Universal Robots PolyScope program: inkscape-test-1.urp

Program inkscape-test-1 (installation=default directory=/programs createdIn=5.11.9.1010452 lastSavedIn=5.11.9.1010452 robotSerialNumber=20225200364)
Calibrated DH parameters: a=[0.00002, -0.569483, -0.54992, -0.00001, -0.000036, 0]; d=[0.180894, -146.691669, 192.918669, -46.053088, 0.119778, 0.115602]; alpha=[1.571425, -0.001534, 0.003359, 1.568739, -1.571477, 0]; deltaTheta=[0, 0.376258, -0.101074, -0.275185, -0.000002, 0]
Robot Program (runOnlyOnce=true)
  Script file /programs/usbdisk/robot_new_inkscape_test_9.script
    | def Machining3():
    |   # Default parameters:
    |   global speed_ms = 0.3
    |   global speed_rads = 0.75
    |   global accel_mss = 3
    |   global accel_radss = 1.2
    |   global blend_radius_m = 0.001
    | 
    |   # Add subprograms here
    |   # Start of main program
    |   # Program generated by RoboDK v5.6.5 for UR10e on 16/10/2023 17:33:41
    |   # Using nominal kinematics.
    |   blend_radius_m = 0.001
    |   speed_ms = 1.000
    |   # set_reference(p[0.335000, -0.154000, -0.015800, 0.000000, 0.000000, 0.000000])
    |   set_tcp(p[0.000000, 0.000000, 0.252000, 0.000000, 0.000000, 0.000000])
    |   # Show Tool
    |   movej([0.061043, -1.073805, -2.582860, -1.055724, 1.570796, 1.631840],accel_radss,speed_rads,0,blend_radius_m)
    |   movel([0.061043, -1.164815, -2.648932, -0.898642, 1.570796, 1.631840],accel_mss,speed_ms,0,blend_radius_m)
    |   speed_ms = 1.000
    |   speed_ms = 0.005
    |   movel([0.061043, -1.124589, -2.623317, -0.964483, 1.570796, 1.631840],accel_mss,speed_ms,0,blend_radius_m)
    |   speed_ms = 1.000
    |   movel([0.061043, -1.164815, -2.648932, -0.898642, 1.570796, 1.631840],accel_mss,speed_ms,0,blend_radius_m)
    |   speed_ms = 0.040
    |   speed_ms = 1.000
    |   movel([0.120277, -1.219092, -2.622470, -0.870827, 1.570796, 1.691073],accel_mss,speed_ms,0,blend_radius_m)
    |   speed_ms = 0.005
    |   movel([0.120277, -1.264094, -2.645638, -0.802657, 1.570796, 1.691073],accel_mss,speed_ms,0,blend_radius_m)
    |   speed_ms = 0.030
    |   movel([0.129753, -1.261000, -2.647334, -0.804055, 1.570796, 1.700549],accel_mss,speed_ms,0,blend_radius_m)
    |   movel([0.141933, -1.256916, -2.649554, -0.805919, 1.570796, 1.712729],accel_mss,speed_ms,0,blend_radius_m)
    |   movel([0.142238, -1.256582, -2.649735, -0.806073, 1.570796, 1.713034],accel_mss,speed_ms,0,blend_radius_m)
    |   movel([0.142012, -1.256413, -2.649826, -0.806150, 1.570796, 1.712808],accel_mss,speed_ms,0,blend_radius_m)
    |   movel([0.136669, -1.257955, -2.648991, -0.805443, 1.570796, 1.707466],accel_mss,speed_ms,0,blend_radius_m)
    |   movel([0.120416, -1.263053, -2.646210, -0.803126, 1.570796, 1.691212],accel_mss,speed_ms,0,blend_radius_m)
    |   movel([0.110953, -1.266208, -2.644473, -0.801708, 1.570796, 1.681749],accel_mss,speed_ms,0,blend_radius_m)
    |   movel([0.098869, -1.270513, -2.642083, -0.799793, 1.570796, 1.669665],accel_mss,speed_ms,0,blend_radius_m)
    |   movel([0.098580, -1.270845, -2.641898, -0.799646, 1.570796, 1.669376],accel_mss,speed_ms,0,blend_radius_m)
    |   movel([0.098815, -1.270997, -2.641813, -0.799579, 1.570796, 1.669612],accel_mss,speed_ms,0,blend_radius_m)
    |   movel([0.104107, -1.269335, -2.642739, -0.800314, 1.570796, 1.674903],accel_mss,speed_ms,0,blend_radius_m)
    |   movel([0.120277, -1.264094, -2.645638, -0.802657, 1.570796, 1.691073],accel_mss,speed_ms,0,blend_radius_m)
    |   movel([0.123150, -1.263148, -2.646158, -0.803083, 1.570796, 1.693947],accel_mss,speed_ms,0,blend_radius_m)
    |   speed_ms = 0.005
    |   movel([0.123150, -1.253718, -2.641632, -0.817039, 1.570796, 1.693947],accel_mss,speed_ms,0,blend_radius_m)
    |   speed_ms = 0.040
    |   movel([0.120555, -1.252576, -2.642250, -0.817563, 1.570796, 1.691351],accel_mss,speed_ms,0,blend_radius_m)
    |   speed_ms = 0.005
    |   movel([0.120555, -1.262011, -2.646781, -0.803597, 1.570796, 1.691351],accel_mss,speed_ms,0,blend_radius_m)
    |   speed_ms = 0.030
    |   movel([0.142487, -1.254991, -2.650593, -0.806805, 1.570796, 1.713283],accel_mss,speed_ms,0,blend_radius_m)
    |   movel([0.142694, -1.253662, -2.651308, -0.807419, 1.570796, 1.713491],accel_mss,speed_ms,0,blend_radius_m)
    |   movel([0.142903, -1.252330, -2.652023, -0.808036, 1.570796, 1.713699],accel_mss,speed_ms,0,blend_radius_m)
    |   movel([0.120905, -1.259399, -2.648206, -0.804783, 1.570796, 1.691701],accel_mss,speed_ms,0,blend_radius_m)
    |   movel([0.099033, -1.266750, -2.644174, -0.801466, 1.570796, 1.669830],accel_mss,speed_ms,0,blend_radius_m)
    |   movel([0.098891, -1.268032, -2.643463, -0.800894, 1.570796, 1.669687],accel_mss,speed_ms,0,blend_radius_m)
    |   movel([0.098749, -1.269312, -2.642752, -0.800325, 1.570796, 1.669546],accel_mss,speed_ms,0,blend_radius_m)
    |   movel([0.120555, -1.262011, -2.646781, -0.803597, 1.570796, 1.691351],accel_mss,speed_ms,0,blend_radius_m)
    |   movel([0.123434, -1.261071, -2.647295, -0.804023, 1.570796, 1.694230],accel_mss,speed_ms,0,blend_radius_m)
    |   speed_ms = 0.005
    |   movel([0.123434, -1.251631, -2.642760, -0.817998, 1.570796, 1.694230],accel_mss,speed_ms,0,blend_radius_m)
    |   speed_ms = 0.040
    |   movel([0.121045, -1.248898, -2.644228, -0.819263, 1.570796, 1.691842],accel_mss,speed_ms,0,blend_radius_m)
    |   speed_ms = 0.005
    |   movel([0.121045, -1.258351, -2.648776, -0.805262, 1.570796, 1.691842],accel_mss,speed_ms,0,blend_radius_m)
    |   speed_ms = 0.030
    |   movel([0.106723, -1.263119, -2.646174, -0.803096, 1.570796, 1.677520],accel_mss,speed_ms,0,blend_radius_m)
    |   movel([0.102037, -1.264600, -2.645360, -0.802429, 1.570796, 1.672833],accel_mss,speed_ms,0,blend_radius_m)
    |   movel([0.099769, -1.265127, -2.645070, -0.802192, 1.570796, 1.670566],accel_mss,speed_ms,0,blend_radius_m)
    |   movel([0.099380, -1.265045, -2.645115, -0.802229, 1.570796, 1.670177],accel_mss,speed_ms,0,blend_radius_m)
    |   movel([0.099262, -1.264692, -2.645309, -0.802388, 1.570796, 1.670058],accel_mss,speed_ms,0,blend_radius_m)
    |   movel([0.099472, -1.264226, -2.645566, -0.802597, 1.570796, 1.670268],accel_mss,speed_ms,0,blend_radius_m)
    |   movel([0.099911, -1.263859, -2.645767, -0.802763, 1.570796, 1.670707],accel_mss,speed_ms,0,blend_radius_m)
    |   movel([0.102241, -1.262808, -2.646345, -0.803237, 1.570796, 1.673038],accel_mss,speed_ms,0,blend_radius_m)
    |   movel([0.106966, -1.261080, -2.647290, -0.804019, 1.570796, 1.677763],accel_mss,speed_ms,0,blend_radius_m)
    |   movel([0.121327, -1.256251, -2.649914, -0.806225, 1.570796, 1.692123],accel_mss,speed_ms,0,blend_radius_m)
    |   movel([0.135738, -1.251578, -2.652425, -0.808386, 1.570796, 1.706534],accel_mss,speed_ms,0,blend_radius_m)
    |   movel([0.140472, -1.250185, -2.653169, -0.809035, 1.570796, 1.711269],accel_mss,speed_ms,0,blend_radius_m)
    |   movel([0.142756, -1.249719, -2.653417, -0.809253, 1.570796, 1.713552],accel_mss,speed_ms,0,blend_radius_m)
    |   movel([0.143139, -1.249820, -2.653363, -0.809206, 1.570796, 1.713935],accel_mss,speed_ms,0,blend_radius_m)
    |   movel([0.143238, -1.250193, -2.653165, -0.809031, 1.570796, 1.714034],accel_mss,speed_ms,0,blend_radius_m)
    |   movel([0.143005, -1.250671, -2.652910, -0.808808, 1.570796, 1.713802],accel_mss,speed_ms,0,blend_radius_m)
    |   movel([0.142550, -1.251035, -2.652715, -0.808639, 1.570796, 1.713347],accel_mss,speed_ms,0,blend_radius_m)
    |   movel([0.140187, -1.252037, -2.652180, -0.808172, 1.570796, 1.710984],accel_mss,speed_ms,0,blend_radius_m)
    |   movel([0.135426, -1.253668, -2.651305, -0.807416, 1.570796, 1.706223],accel_mss,speed_ms,0,blend_radius_m)
    |   movel([0.121045, -1.258351, -2.648776, -0.805262, 1.570796, 1.691842],accel_mss,speed_ms,0,blend_radius_m)
    |   movel([0.118157, -1.259303, -2.648259, -0.804827, 1.570796, 1.688953],accel_mss,speed_ms,0,blend_radius_m)
    |   speed_ms = 0.005
    |   movel([0.118157, -1.249854, -2.643716, -0.818819, 1.570796, 1.688953],accel_mss,speed_ms,0,blend_radius_m)
    |   speed_ms = 0.040
    |   movel([0.121469, -1.245729, -2.645920, -0.820740, 1.570796, 1.692265],accel_mss,speed_ms,0,blend_radius_m)
    |   speed_ms = 0.005
    |   movel([0.121469, -1.255197, -2.650482, -0.806710, 1.570796, 1.692265],accel_mss,speed_ms,0,blend_radius_m)
    |   speed_ms = 0.030
    |   movel([0.105133, -1.260563, -2.647572, -0.804254, 1.570796, 1.675929],accel_mss,speed_ms,0,blend_radius_m)
    |   movel([0.099787, -1.262265, -2.646642, -0.803482, 1.570796, 1.670583],accel_mss,speed_ms,0,blend_radius_m)
    |   movel([0.099549, -1.262111, -2.646726, -0.803552, 1.570796, 1.670346],accel_mss,speed_ms,0,blend_radius_m)
    |   movel([0.099842, -1.261774, -2.646911, -0.803704, 1.570796, 1.670638],accel_mss,speed_ms,0,blend_radius_m)
    |   movel([0.112050, -1.257371, -2.649308, -0.805711, 1.570796, 1.682846],accel_mss,speed_ms,0,blend_radius_m)
    |   movel([0.121610, -1.254143, -2.651050, -0.807196, 1.570796, 1.692407],accel_mss,speed_ms,0,blend_radius_m)
    |   movel([0.138032, -1.248922, -2.653841, -0.809626, 1.570796, 1.708829],accel_mss,speed_ms,0,blend_radius_m)
    |   movel([0.143430, -1.247342, -2.654680, -0.810368, 1.570796, 1.714226],accel_mss,speed_ms,0,blend_radius_m)
    |   movel([0.143659, -1.247512, -2.654589, -0.810288, 1.570796, 1.714455],accel_mss,speed_ms,0,blend_radius_m)
    |   movel([0.143350, -1.247852, -2.654409, -0.810128, 1.570796, 1.714146],accel_mss,speed_ms,0,blend_radius_m)
    |   movel([0.131042, -1.252031, -2.652183, -0.808175, 1.570796, 1.701839],accel_mss,speed_ms,0,blend_radius_m)
    |   movel([0.121469, -1.255197, -2.650482, -0.806710, 1.570796, 1.692265],accel_mss,speed_ms,0,blend_radius_m)
    |   movel([0.118572, -1.256136, -2.649976, -0.806278, 1.570796, 1.689369],accel_mss,speed_ms,0,blend_radius_m)
    |   speed_ms = 0.005
    |   movel([0.118572, -1.246672, -2.645418, -0.820299, 1.570796, 1.689369],accel_mss,speed_ms,0,blend_radius_m)
    |   speed_ms = 0.040
    |   movel([0.121895, -1.242544, -2.647608, -0.822237, 1.570796, 1.692691],accel_mss,speed_ms,0,blend_radius_m)
    |   speed_ms = 0.005
    |   movel([0.121895, -1.252028, -2.652185, -0.808177, 1.570796, 1.692691],accel_mss,speed_ms,0,blend_radius_m)
    |   speed_ms = 0.030
    |   movel([0.099260, -1.259721, -2.648031, -0.804637, 1.570796, 1.670056],accel_mss,speed_ms,0,blend_radius_m)
    |   movel([0.101199, -1.242362, -2.657302, -0.812725, 1.570796, 1.671995],accel_mss,speed_ms,0,blend_radius_m)
    |   movel([0.103217, -1.224523, -2.666459, -0.821407, 1.570796, 1.674013],accel_mss,speed_ms,0,blend_radius_m)
    |   movel([0.126797, -1.216082, -2.670663, -0.825644, 1.570796, 1.697593],accel_mss,speed_ms,0,blend_radius_m)
    |   movel([0.150532, -1.207955, -2.674635, -0.829799, 1.570796, 1.721329],accel_mss,speed_ms,0,blend_radius_m)
    |   movel([0.147540, -1.226560, -2.665432, -0.820397, 1.570796, 1.718336],accel_mss,speed_ms,0,blend_radius_m)
    |   movel([0.144667, -1.244634, -2.656110, -0.811646, 1.570796, 1.715464],accel_mss,speed_ms,0,blend_radius_m)
    |   movel([0.121895, -1.252028, -2.652185, -0.808177, 1.570796, 1.692691],accel_mss,speed_ms,0,blend_radius_m)
    |   movel([0.118985, -1.252998, -2.651665, -0.807726, 1.570796, 1.689781],accel_mss,speed_ms,0,blend_radius_m)
    |   speed_ms = 0.005
    |   movel([0.118985, -1.243519, -2.647093, -0.821777, 1.570796, 1.689781],accel_mss,speed_ms,0,blend_radius_m)
    |   speed_ms = 0.040
    |   movel([0.126726, -1.204862, -2.666692, -0.840834, 1.570796, 1.697522],accel_mss,speed_ms,0,blend_radius_m)
    |   speed_ms = 0.005
    |   movel([0.126726, -1.214506, -2.671439, -0.826444, 1.570796, 1.697522],accel_mss,speed_ms,0,blend_radius_m)
    |   speed_ms = 0.030
    |   movel([0.104008, -1.222655, -2.667396, -0.822338, 1.570796, 1.674804],accel_mss,speed_ms,0,blend_radius_m)
    |   movel([0.105123, -1.212962, -2.672197, -0.827230, 1.570796, 1.675919],accel_mss,speed_ms,0,blend_radius_m)
    |   movel([0.106263, -1.203120, -2.676963, -0.832306, 1.570796, 1.677059],accel_mss,speed_ms,0,blend_radius_m)
    |   movel([0.129497, -1.194544, -2.681029, -0.836816, 1.570796, 1.700293],accel_mss,speed_ms,0,blend_radius_m)
    |   movel([0.152886, -1.186265, -2.684878, -0.841246, 1.570796, 1.723683],accel_mss,speed_ms,0,blend_radius_m)
    |   movel([0.151219, -1.196537, -2.680091, -0.835761, 1.570796, 1.722015],accel_mss,speed_ms,0,blend_radius_m)
    |   movel([0.149588, -1.206647, -2.675268, -0.830475, 1.570796, 1.720384],accel_mss,speed_ms,0,blend_radius_m)
    |   movel([0.126726, -1.214506, -2.671439, -0.826444, 1.570796, 1.697522],accel_mss,speed_ms,0,blend_radius_m)
    |   movel([0.123688, -1.215576, -2.670913, -0.825900, 1.570796, 1.694484],accel_mss,speed_ms,0,blend_radius_m)
    |   speed_ms = 0.005
    |   movel([0.123688, -1.205937, -2.666170, -0.840282, 1.570796, 1.694484],accel_mss,speed_ms,0,blend_radius_m)
    |   speed_ms = 0.040
    |   movel([0.157276, -1.164256, -2.685501, -0.862631, 1.570796, 1.728073],accel_mss,speed_ms,0,blend_radius_m)
    |   speed_ms = 0.005
    |   movel([0.157276, -1.174031, -2.690432, -0.847927, 1.570796, 1.728073],accel_mss,speed_ms,0,blend_radius_m)
    |   speed_ms = 0.030
    |   movel([0.255784, -1.142912, -2.703858, -0.865619, 1.570796, 1.826580],accel_mss,speed_ms,0,blend_radius_m)
    |   movel([0.213690, -1.314067, -2.616588, -0.781734, 1.570796, 1.784487],accel_mss,speed_ms,0,blend_radius_m)
    |   movel([0.183803, -1.448210, -2.521691, -0.742489, 1.570796, 1.754599],accel_mss,speed_ms,0,blend_radius_m)
    |   movel([0.113774, -1.462570, -2.509956, -0.739863, 1.570796, 1.684571],accel_mss,speed_ms,0,blend_radius_m)
    |   movel([0.044558, -1.480296, -2.495031, -0.737062, 1.570796, 1.615354],accel_mss,speed_ms,0,blend_radius_m)
    |   movel([0.051500, -1.358795, -2.587796, -0.765798, 1.570796, 1.622297],accel_mss,speed_ms,0,blend_radius_m)
    |   movel([0.061043, -1.210716, -2.673294, -0.828379, 1.570796, 1.631840],accel_mss,speed_ms,0,blend_radius_m)
    |   movel([0.157276, -1.174031, -2.690432, -0.847927, 1.570796, 1.728073],accel_mss,speed_ms,0,blend_radius_m)
    |   movel([0.160447, -1.172924, -2.690926, -0.848539, 1.570796, 1.731244],accel_mss,speed_ms,0,blend_radius_m)
    |   speed_ms = 0.005
    |   movel([0.160447, -1.163146, -2.685991, -0.863252, 1.570796, 1.731244],accel_mss,speed_ms,0,blend_radius_m)
    |   speed_ms = 0.040
    |   movel([0.178723, -1.187438, -2.674979, -0.849972, 1.570796, 1.749519],accel_mss,speed_ms,0,blend_radius_m)
    |   speed_ms = 0.005
    |   movel([0.178723, -1.197143, -2.679805, -0.835441, 1.570796, 1.749519],accel_mss,speed_ms,0,blend_radius_m)
    |   speed_ms = 0.030
    |   movel([0.155706, -1.204603, -2.676252, -0.831534, 1.570796, 1.726503],accel_mss,speed_ms,0,blend_radius_m)
    |   movel([0.157407, -1.194439, -2.681078, -0.836872, 1.570796, 1.728204],accel_mss,speed_ms,0,blend_radius_m)
    |   movel([0.159147, -1.184110, -2.685868, -0.842411, 1.570796, 1.729943],accel_mss,speed_ms,0,blend_radius_m)
    |   movel([0.182702, -1.176243, -2.689439, -0.846707, 1.570796, 1.753498],accel_mss,speed_ms,0,blend_radius_m)
    |   movel([0.206362, -1.168729, -2.692789, -0.850871, 1.570796, 1.777158],accel_mss,speed_ms,0,blend_radius_m)
    |   movel([0.204073, -1.179467, -2.687983, -0.844938, 1.570796, 1.774869],accel_mss,speed_ms,0,blend_radius_m)
    |   movel([0.201836, -1.190024, -2.683139, -0.839225, 1.570796, 1.772633],accel_mss,speed_ms,0,blend_radius_m)
    |   movel([0.178723, -1.197143, -2.679805, -0.835441, 1.570796, 1.749519],accel_mss,speed_ms,0,blend_radius_m)
    |   movel([0.175648, -1.198119, -2.679344, -0.834926, 1.570796, 1.746444],accel_mss,speed_ms,0,blend_radius_m)
    |   speed_ms = 0.005
    |   movel([0.175648, -1.188417, -2.674523, -0.849450, 1.570796, 1.746444],accel_mss,speed_ms,0,blend_radius_m)
    |   speed_ms = 0.040
    |   movel([0.170964, -1.226858, -2.655750, -0.829781, 1.570796, 1.741760],accel_mss,speed_ms,0,blend_radius_m)
    |   speed_ms = 0.005
    |   movel([0.170964, -1.236412, -2.660397, -0.815579, 1.570796, 1.741760],accel_mss,speed_ms,0,blend_radius_m)
    |   speed_ms = 0.030
    |   movel([0.193490, -1.230002, -2.663685, -0.818701, 1.570796, 1.764287],accel_mss,speed_ms,0,blend_radius_m)
    |   movel([0.197334, -1.211473, -2.672925, -0.827991, 1.570796, 1.768131],accel_mss,speed_ms,0,blend_radius_m)
    |   movel([0.199301, -1.201920, -2.677537, -0.832932, 1.570796, 1.770097],accel_mss,speed_ms,0,blend_radius_m)
    |   movel([0.200933, -1.192747, -2.681871, -0.837771, 1.570796, 1.771729],accel_mss,speed_ms,0,blend_radius_m)
    |   movel([0.200878, -1.192448, -2.682010, -0.837931, 1.570796, 1.771674],accel_mss,speed_ms,0,blend_radius_m)
    |   movel([0.200628, -1.192319, -2.682071, -0.837999, 1.570796, 1.771424],accel_mss,speed_ms,0,blend_radius_m)
    |   movel([0.200026, -1.192393, -2.682036, -0.837960, 1.570796, 1.770823],accel_mss,speed_ms,0,blend_radius_m)
    |   movel([0.177133, -1.199429, -2.678723, -0.834237, 1.570796, 1.747930],accel_mss,speed_ms,0,blend_radius_m)
    |   movel([0.154454, -1.206920, -2.675136, -0.830334, 1.570796, 1.725251],accel_mss,speed_ms,0,blend_radius_m)
    |   movel([0.151426, -1.225300, -2.666067, -0.821021, 1.570796, 1.722223],accel_mss,speed_ms,0,blend_radius_m)
    |   movel([0.148519, -1.243161, -2.656883, -0.812345, 1.570796, 1.719315],accel_mss,speed_ms,0,blend_radius_m)
    |   movel([0.170964, -1.236412, -2.660397, -0.815579, 1.570796, 1.741760],accel_mss,speed_ms,0,blend_radius_m)
    |   movel([0.173904, -1.235555, -2.660840, -0.815994, 1.570796, 1.744701],accel_mss,speed_ms,0,blend_radius_m)
    |   speed_ms = 0.005
    |   movel([0.173904, -1.225997, -2.656189, -0.830203, 1.570796, 1.744701],accel_mss,speed_ms,0,blend_radius_m)
    |   speed_ms = 0.040
    |   movel([0.170186, -1.230349, -2.653963, -0.828077, 1.570796, 1.740982],accel_mss,speed_ms,0,blend_radius_m)
    |   speed_ms = 0.005
    |   movel([0.170186, -1.239888, -2.658594, -0.813906, 1.570796, 1.740982],accel_mss,speed_ms,0,blend_radius_m)
    |   speed_ms = 0.030
    |   movel([0.182708, -1.236197, -2.660509, -0.815683, 1.570796, 1.753504],accel_mss,speed_ms,0,blend_radius_m)
    |   movel([0.188419, -1.234448, -2.661410, -0.816531, 1.570796, 1.759215],accel_mss,speed_ms,0,blend_radius_m)
    |   movel([0.191800, -1.233306, -2.661997, -0.817086, 1.570796, 1.762597],accel_mss,speed_ms,0,blend_radius_m)
    |   movel([0.192177, -1.233050, -2.662128, -0.817211, 1.570796, 1.762974],accel_mss,speed_ms,0,blend_radius_m)
    |   movel([0.192385, -1.232674, -2.662321, -0.817394, 1.570796, 1.763181],accel_mss,speed_ms,0,blend_radius_m)
    |   movel([0.192316, -1.232375, -2.662474, -0.817540, 1.570796, 1.763112],accel_mss,speed_ms,0,blend_radius_m)
    |   movel([0.192004, -1.232313, -2.662506, -0.817570, 1.570796, 1.762800],accel_mss,speed_ms,0,blend_radius_m)
    |   movel([0.188697, -1.233067, -2.662119, -0.817203, 1.570796, 1.759494],accel_mss,speed_ms,0,blend_radius_m)
    |   movel([0.183024, -1.234583, -2.661341, -0.816465, 1.570796, 1.753821],accel_mss,speed_ms,0,blend_radius_m)
    |   movel([0.170489, -1.238241, -2.659451, -0.814698, 1.570796, 1.741285],accel_mss,speed_ms,0,blend_radius_m)
    |   movel([0.157971, -1.242050, -2.657466, -0.812873, 1.570796, 1.728768],accel_mss,speed_ms,0,blend_radius_m)
    |   movel([0.152285, -1.243917, -2.656487, -0.811986, 1.570796, 1.723081],accel_mss,speed_ms,0,blend_radius_m)
    |   movel([0.148931, -1.245142, -2.655842, -0.811405, 1.570796, 1.719727],accel_mss,speed_ms,0,blend_radius_m)
    |   movel([0.148564, -1.245403, -2.655704, -0.811282, 1.570796, 1.719360],accel_mss,speed_ms,0,blend_radius_m)
    |   movel([0.148374, -1.245773, -2.655509, -0.811107, 1.570796, 1.719170],accel_mss,speed_ms,0,blend_radius_m)
    |   movel([0.148458, -1.246056, -2.655359, -0.810973, 1.570796, 1.719254],accel_mss,speed_ms,0,blend_radius_m)
    |   movel([0.148775, -1.246103, -2.655335, -0.810951, 1.570796, 1.719571],accel_mss,speed_ms,0,blend_radius_m)
    |   movel([0.152063, -1.245259, -2.655780, -0.811350, 1.570796, 1.722859],accel_mss,speed_ms,0,blend_radius_m)
    |   movel([0.157700, -1.243633, -2.656636, -0.812120, 1.570796, 1.728496],accel_mss,speed_ms,0,blend_radius_m)
    |   movel([0.170186, -1.239888, -2.658594, -0.813906, 1.570796, 1.740982],accel_mss,speed_ms,0,blend_radius_m)
    |   movel([0.173119, -1.239014, -2.659049, -0.814326, 1.570796, 1.743916],accel_mss,speed_ms,0,blend_radius_m)
    |   speed_ms = 0.005
    |   movel([0.173119, -1.229471, -2.654414, -0.828505, 1.570796, 1.743916],accel_mss,speed_ms,0,blend_radius_m)
    |   speed_ms = 0.040
    |   movel([0.169583, -1.233646, -2.652262, -0.826481, 1.570796, 1.740380],accel_mss,speed_ms,0,blend_radius_m)
    |   speed_ms = 0.005
    |   movel([0.169583, -1.243171, -2.656878, -0.812340, 1.570796, 1.740380],accel_mss,speed_ms,0,blend_radius_m)
    |   speed_ms = 0.030
    |   movel([0.155296, -1.247453, -2.654621, -0.810316, 1.570796, 1.726092],accel_mss,speed_ms,0,blend_radius_m)
    |   movel([0.150619, -1.248774, -2.653920, -0.809695, 1.570796, 1.721416],accel_mss,speed_ms,0,blend_radius_m)
    |   movel([0.148370, -1.249213, -2.653686, -0.809489, 1.570796, 1.719166],accel_mss,speed_ms,0,blend_radius_m)
    |   movel([0.147989, -1.249108, -2.653742, -0.809539, 1.570796, 1.718786],accel_mss,speed_ms,0,blend_radius_m)
    |   movel([0.147895, -1.248734, -2.653941, -0.809714, 1.570796, 1.718691],accel_mss,speed_ms,0,blend_radius_m)
    |   movel([0.148126, -1.248259, -2.654193, -0.809937, 1.570796, 1.718923],accel_mss,speed_ms,0,blend_radius_m)
    |   movel([0.148584, -1.247891, -2.654388, -0.810109, 1.570796, 1.719381],accel_mss,speed_ms,0,blend_radius_m)
    |   movel([0.150927, -1.246905, -2.654911, -0.810573, 1.570796, 1.721723],accel_mss,speed_ms,0,blend_radius_m)
    |   movel([0.155655, -1.245329, -2.655743, -0.811317, 1.570796, 1.726451],accel_mss,speed_ms,0,blend_radius_m)
    |   movel([0.169984, -1.240984, -2.658023, -0.813382, 1.570796, 1.740781],accel_mss,speed_ms,0,blend_radius_m)
    |   movel([0.184343, -1.236813, -2.660190, -0.815386, 1.570796, 1.755139],accel_mss,speed_ms,0,blend_radius_m)
    |   movel([0.189052, -1.235591, -2.660821, -0.815976, 1.570796, 1.759849],accel_mss,speed_ms,0,blend_radius_m)
    |   movel([0.191309, -1.235219, -2.661013, -0.816157, 1.570796, 1.762105],accel_mss,speed_ms,0,blend_radius_m)
    |   movel([0.191682, -1.235344, -2.660949, -0.816096, 1.570796, 1.762478],accel_mss,speed_ms,0,blend_radius_m)
    |   movel([0.191756, -1.235737, -2.660746, -0.815906, 1.570796, 1.762552],accel_mss,speed_ms,0,blend_radius_m)
    |   movel([0.191502, -1.236222, -2.660496, -0.815671, 1.570796, 1.762298],accel_mss,speed_ms,0,blend_radius_m)
    |   movel([0.191030, -1.236585, -2.660308, -0.815496, 1.570796, 1.761826],accel_mss,speed_ms,0,blend_radius_m)
    |   movel([0.188663, -1.237515, -2.659827, -0.815047, 1.570796, 1.759460],accel_mss,speed_ms,0,blend_radius_m)
    |   movel([0.183914, -1.238984, -2.659064, -0.814340, 1.570796, 1.754710],accel_mss,speed_ms,0,blend_radius_m)
    |   movel([0.169583, -1.243171, -2.656878, -0.812340, 1.570796, 1.740380],accel_mss,speed_ms,0,blend_radius_m)
    |   movel([0.166664, -1.244035, -2.656424, -0.811929, 1.570796, 1.737460],accel_mss,speed_ms,0,blend_radius_m)
    |   speed_ms = 0.005
    |   movel([0.166664, -1.234514, -2.651812, -0.826063, 1.570796, 1.737460],accel_mss,speed_ms,0,blend_radius_m)
    |   speed_ms = 0.040
    |   movel([0.168985, -1.236926, -2.650557, -0.824906, 1.570796, 1.739782],accel_mss,speed_ms,0,blend_radius_m)
    |   speed_ms = 0.005
    |   movel([0.168985, -1.246436, -2.655159, -0.810794, 1.570796, 1.739782],accel_mss,speed_ms,0,blend_radius_m)
    |   speed_ms = 0.030
    |   movel([0.154750, -1.250681, -2.652904, -0.808803, 1.570796, 1.725547],accel_mss,speed_ms,0,blend_radius_m)
    |   movel([0.150091, -1.251991, -2.652204, -0.808194, 1.570796, 1.720887],accel_mss,speed_ms,0,blend_radius_m)
    |   movel([0.147850, -1.252426, -2.651971, -0.807991, 1.570796, 1.718646],accel_mss,speed_ms,0,blend_radius_m)
    |   movel([0.147470, -1.252321, -2.652028, -0.808041, 1.570796, 1.718267],accel_mss,speed_ms,0,blend_radius_m)
    |   movel([0.147376, -1.251949, -2.652227, -0.808213, 1.570796, 1.718172],accel_mss,speed_ms,0,blend_radius_m)
    |   movel([0.147607, -1.251476, -2.652480, -0.808433, 1.570796, 1.718403],accel_mss,speed_ms,0,blend_radius_m)
    |   movel([0.148063, -1.251111, -2.652675, -0.808603, 1.570796, 1.718859],accel_mss,speed_ms,0,blend_radius_m)
    |   movel([0.150396, -1.250132, -2.653197, -0.809060, 1.570796, 1.721192],accel_mss,speed_ms,0,blend_radius_m)
    |   movel([0.155107, -1.248568, -2.654029, -0.809792, 1.570796, 1.725903],accel_mss,speed_ms,0,blend_radius_m)
    |   movel([0.169384, -1.244261, -2.656306, -0.811822, 1.570796, 1.740180],accel_mss,speed_ms,0,blend_radius_m)
    |   movel([0.183688, -1.240125, -2.658471, -0.813793, 1.570796, 1.754485],accel_mss,speed_ms,0,blend_radius_m)
    |   movel([0.188381, -1.238915, -2.659101, -0.814374, 1.570796, 1.759177],accel_mss,speed_ms,0,blend_radius_m)
    |   movel([0.190629, -1.238546, -2.659292, -0.814551, 1.570796, 1.761425],accel_mss,speed_ms,0,blend_radius_m)
    |   movel([0.191001, -1.238672, -2.659227, -0.814490, 1.570796, 1.761797],accel_mss,speed_ms,0,blend_radius_m)
    |   movel([0.191075, -1.239063, -2.659024, -0.814303, 1.570796, 1.761871],accel_mss,speed_ms,0,blend_radius_m)
    |   movel([0.190822, -1.239545, -2.658773, -0.814071, 1.570796, 1.761618],accel_mss,speed_ms,0,blend_radius_m)
    |   movel([0.190352, -1.239905, -2.658585, -0.813898, 1.570796, 1.761148],accel_mss,speed_ms,0,blend_radius_m)
    |   movel([0.187994, -1.240828, -2.658104, -0.813456, 1.570796, 1.758791],accel_mss,speed_ms,0,blend_radius_m)
    |   movel([0.183262, -1.242285, -2.657342, -0.812761, 1.570796, 1.754059],accel_mss,speed_ms,0,blend_radius_m)
    |   movel([0.168985, -1.246436, -2.655159, -0.810794, 1.570796, 1.739782],accel_mss,speed_ms,0,blend_radius_m)
    |   movel([0.166076, -1.247293, -2.654706, -0.810391, 1.570796, 1.736873],accel_mss,speed_ms,0,blend_radius_m)
    |   speed_ms = 0.005
    |   movel([0.166076, -1.237787, -2.650108, -0.824494, 1.570796, 1.736873],accel_mss,speed_ms,0,blend_radius_m)
    |   speed_ms = 0.040
    |   movel([0.168490, -1.239647, -2.649134, -0.823609, 1.570796, 1.739287],accel_mss,speed_ms,0,blend_radius_m)
    |   speed_ms = 0.005
    |   movel([0.168490, -1.249144, -2.653723, -0.809522, 1.570796, 1.739287],accel_mss,speed_ms,0,blend_radius_m)
    |   speed_ms = 0.030
    |   movel([0.156135, -1.252799, -2.651772, -0.807819, 1.570796, 1.726931],accel_mss,speed_ms,0,blend_radius_m)
    |   movel([0.150556, -1.254386, -2.650919, -0.807084, 1.570796, 1.721352],accel_mss,speed_ms,0,blend_radius_m)
    |   movel([0.147302, -1.255208, -2.650476, -0.806704, 1.570796, 1.718098],accel_mss,speed_ms,0,blend_radius_m)
    |   movel([0.146988, -1.255161, -2.650502, -0.806726, 1.570796, 1.717784],accel_mss,speed_ms,0,blend_radius_m)
    |   movel([0.146904, -1.254881, -2.650652, -0.806855, 1.570796, 1.717700],accel_mss,speed_ms,0,blend_radius_m)
    |   movel([0.147092, -1.254517, -2.650848, -0.807023, 1.570796, 1.717888],accel_mss,speed_ms,0,blend_radius_m)
    |   movel([0.147454, -1.254261, -2.650986, -0.807142, 1.570796, 1.718251],accel_mss,speed_ms,0,blend_radius_m)
    |   movel([0.150774, -1.253063, -2.651630, -0.807696, 1.570796, 1.721570],accel_mss,speed_ms,0,blend_radius_m)
    |   movel([0.156400, -1.251239, -2.652606, -0.808543, 1.570796, 1.727197],accel_mss,speed_ms,0,blend_radius_m)
    |   movel([0.168787, -1.247520, -2.654585, -0.810284, 1.570796, 1.739583],accel_mss,speed_ms,0,blend_radius_m)
    |   movel([0.181191, -1.243951, -2.656469, -0.811969, 1.570796, 1.751988],accel_mss,speed_ms,0,blend_radius_m)
    |   movel([0.186805, -1.242473, -2.657244, -0.812672, 1.570796, 1.757601],accel_mss,speed_ms,0,blend_radius_m)
    |   movel([0.190077, -1.241738, -2.657629, -0.813022, 1.570796, 1.760873],accel_mss,speed_ms,0,blend_radius_m)
    |   movel([0.190386, -1.241800, -2.657596, -0.812992, 1.570796, 1.761182],accel_mss,speed_ms,0,blend_radius_m)
    |   movel([0.190455, -1.242095, -2.657442, -0.812852, 1.570796, 1.761251],accel_mss,speed_ms,0,blend_radius_m)
    |   movel([0.190250, -1.242466, -2.657248, -0.812675, 1.570796, 1.761047],accel_mss,speed_ms,0,blend_radius_m)
    |   movel([0.189878, -1.242717, -2.657116, -0.812556, 1.570796, 1.760674],accel_mss,speed_ms,0,blend_radius_m)
    |   movel([0.186532, -1.243833, -2.656531, -0.812025, 1.570796, 1.757329],accel_mss,speed_ms,0,blend_radius_m)
    |   movel([0.180881, -1.245540, -2.655632, -0.811217, 1.570796, 1.751678],accel_mss,speed_ms,0,blend_radius_m)
    |   movel([0.168490, -1.249144, -2.653723, -0.809522, 1.570796, 1.739287],accel_mss,speed_ms,0,blend_radius_m)
    |   movel([0.165591, -1.249992, -2.653272, -0.809125, 1.570796, 1.736387],accel_mss,speed_ms,0,blend_radius_m)
    |   speed_ms = 0.005
    |   movel([0.165591, -1.240499, -2.648686, -0.823204, 1.570796, 1.736387],accel_mss,speed_ms,0,blend_radius_m)
    |   speed_ms = 0.040
    |   movel([0.159403, -1.290501, -2.620887, -0.801001, 1.570796, 1.730199],accel_mss,speed_ms,0,blend_radius_m)
    |   speed_ms = 0.005
    |   movel([0.159403, -1.299735, -2.625247, -0.787408, 1.570796, 1.730199],accel_mss,speed_ms,0,blend_radius_m)
    |   speed_ms = 0.030
    |   movel([0.138633, -1.305540, -2.621772, -0.785077, 1.570796, 1.709430],accel_mss,speed_ms,0,blend_radius_m)
    |   movel([0.142308, -1.282036, -2.635573, -0.794780, 1.570796, 1.713104],accel_mss,speed_ms,0,blend_radius_m)
    |   movel([0.146189, -1.257624, -2.649170, -0.805595, 1.570796, 1.716985],accel_mss,speed_ms,0,blend_radius_m)
    |   movel([0.167590, -1.251060, -2.652702, -0.808627, 1.570796, 1.738386],accel_mss,speed_ms,0,blend_radius_m)
    |   movel([0.189184, -1.244915, -2.655961, -0.811513, 1.570796, 1.759980],accel_mss,speed_ms,0,blend_radius_m)
    |   movel([0.189757, -1.244857, -2.655992, -0.811540, 1.570796, 1.760554],accel_mss,speed_ms,0,blend_radius_m)
    |   movel([0.190007, -1.244989, -2.655922, -0.811478, 1.570796, 1.760803],accel_mss,speed_ms,0,blend_radius_m)
    |   movel([0.190058, -1.245287, -2.655765, -0.811337, 1.570796, 1.760855],accel_mss,speed_ms,0,blend_radius_m)
    |   movel([0.187829, -1.257249, -2.649373, -0.805766, 1.570796, 1.758625],accel_mss,speed_ms,0,blend_radius_m)
    |   movel([0.185199, -1.270058, -2.642337, -0.799994, 1.570796, 1.755995],accel_mss,speed_ms,0,blend_radius_m)
    |   movel([0.180242, -1.294220, -2.628507, -0.789662, 1.570796, 1.751038],accel_mss,speed_ms,0,blend_radius_m)
    |   movel([0.159403, -1.299735, -2.625247, -0.787408, 1.570796, 1.730199],accel_mss,speed_ms,0,blend_radius_m)
    |   movel([0.156666, -1.300482, -2.624802, -0.787105, 1.570796, 1.727462],accel_mss,speed_ms,0,blend_radius_m)
    |   speed_ms = 0.005
    |   movel([0.156666, -1.291253, -2.620446, -0.800691, 1.570796, 1.727462],accel_mss,speed_ms,0,blend_radius_m)
    |   speed_ms = 0.040
    |   movel([0.173092, -1.308235, -2.610277, -0.793876, 1.570796, 1.743888],accel_mss,speed_ms,0,blend_radius_m)
    |   speed_ms = 0.005
    |   movel([0.173092, -1.317365, -2.614557, -0.780467, 1.570796, 1.743888],accel_mss,speed_ms,0,blend_radius_m)
    |   speed_ms = 0.030
    |   movel([0.172750, -1.317314, -2.614589, -0.780486, 1.570796, 1.743547],accel_mss,speed_ms,0,blend_radius_m)
    |   movel([0.165825, -1.318972, -2.613562, -0.779854, 1.570796, 1.736621],accel_mss,speed_ms,0,blend_radius_m)
    |   movel([0.148824, -1.323334, -2.610845, -0.778210, 1.570796, 1.719620],accel_mss,speed_ms,0,blend_radius_m)
    |   movel([0.124966, -1.329939, -2.606682, -0.775768, 1.570796, 1.695762],accel_mss,speed_ms,0,blend_radius_m)
    |   movel([0.124236, -1.335108, -2.603382, -0.773898, 1.570796, 1.695032],accel_mss,speed_ms,0,blend_radius_m)
    |   movel([0.148189, -1.328412, -2.607650, -0.776327, 1.570796, 1.718985],accel_mss,speed_ms,0,blend_radius_m)
    |   movel([0.172245, -1.322097, -2.611618, -0.778674, 1.570796, 1.743042],accel_mss,speed_ms,0,blend_radius_m)
    |   movel([0.172824, -1.319862, -2.613010, -0.779517, 1.570796, 1.743620],accel_mss,speed_ms,0,blend_radius_m)
    |   movel([0.173142, -1.318202, -2.614039, -0.780147, 1.570796, 1.743939],accel_mss,speed_ms,0,blend_radius_m)
    |   movel([0.173183, -1.317581, -2.614424, -0.780384, 1.570796, 1.743979],accel_mss,speed_ms,0,blend_radius_m)
    |   movel([0.173092, -1.317365, -2.614557, -0.780467, 1.570796, 1.743888],accel_mss,speed_ms,0,blend_radius_m)
    |   movel([0.172750, -1.317314, -2.614589, -0.780486, 1.570796, 1.743547],accel_mss,speed_ms,0,blend_radius_m)
    |   movel([0.170483, -1.317852, -2.614256, -0.780281, 1.570796, 1.741279],accel_mss,speed_ms,0,blend_radius_m)
    |   speed_ms = 0.005
    |   movel([0.170483, -1.308725, -2.609978, -0.793685, 1.570796, 1.741279],accel_mss,speed_ms,0,blend_radius_m)
    |   speed_ms = 0.040
    |   movel([0.171885, -1.314572, -2.606388, -0.791430, 1.570796, 1.742681],accel_mss,speed_ms,0,blend_radius_m)
    |   speed_ms = 0.005
    |   movel([0.171885, -1.323663, -2.610639, -0.778087, 1.570796, 1.742681],accel_mss,speed_ms,0,blend_radius_m)
    |   speed_ms = 0.030
    |   movel([0.171974, -1.323887, -2.610499, -0.778003, 1.570796, 1.742770],accel_mss,speed_ms,0,blend_radius_m)
    |   movel([0.171923, -1.324565, -2.610074, -0.777750, 1.570796, 1.742719],accel_mss,speed_ms,0,blend_radius_m)
    |   movel([0.171576, -1.326375, -2.608936, -0.777078, 1.570796, 1.742373],accel_mss,speed_ms,0,blend_radius_m)
    |   movel([0.170960, -1.328829, -2.607386, -0.776174, 1.570796, 1.741756],accel_mss,speed_ms,0,blend_radius_m)
    |   movel([0.147241, -1.334878, -2.603531, -0.773981, 1.570796, 1.718037],accel_mss,speed_ms,0,blend_radius_m)
    |   movel([0.123616, -1.341303, -2.599381, -0.771705, 1.570796, 1.694412],accel_mss,speed_ms,0,blend_radius_m)
    |   movel([0.124053, -1.336048, -2.602779, -0.773562, 1.570796, 1.694849],accel_mss,speed_ms,0,blend_radius_m)
    |   movel([0.147766, -1.329542, -2.606934, -0.775913, 1.570796, 1.718562],accel_mss,speed_ms,0,blend_radius_m)
    |   movel([0.164662, -1.325247, -2.609646, -0.777497, 1.570796, 1.735458],accel_mss,speed_ms,0,blend_radius_m)
    |   movel([0.171545, -1.323614, -2.610670, -0.778105, 1.570796, 1.742342],accel_mss,speed_ms,0,blend_radius_m)
    |   movel([0.171885, -1.323663, -2.610639, -0.778087, 1.570796, 1.742681],accel_mss,speed_ms,0,blend_radius_m)
    |   movel([0.171974, -1.323887, -2.610499, -0.778003, 1.570796, 1.742770],accel_mss,speed_ms,0,blend_radius_m)
    |   movel([0.171923, -1.324565, -2.610074, -0.777750, 1.570796, 1.742719],accel_mss,speed_ms,0,blend_radius_m)
    |   movel([0.171652, -1.325981, -2.609184, -0.777224, 1.570796, 1.742448],accel_mss,speed_ms,0,blend_radius_m)
    |   speed_ms = 0.005
    |   movel([0.171652, -1.316905, -2.604942, -0.790542, 1.570796, 1.742448],accel_mss,speed_ms,0,blend_radius_m)
    |   speed_ms = 0.040
    |   movel([0.170695, -1.320851, -2.602481, -0.789057, 1.570796, 1.741491],accel_mss,speed_ms,0,blend_radius_m)
    |   speed_ms = 0.005
    |   movel([0.170695, -1.329903, -2.606705, -0.775781, 1.570796, 1.741491],accel_mss,speed_ms,0,blend_radius_m)
    |   speed_ms = 0.030
    |   movel([0.170785, -1.330115, -2.606570, -0.775704, 1.570796, 1.741581],accel_mss,speed_ms,0,blend_radius_m)
    |   movel([0.170747, -1.330725, -2.606183, -0.775481, 1.570796, 1.741543],accel_mss,speed_ms,0,blend_radius_m)
    |   movel([0.170437, -1.332352, -2.605147, -0.774891, 1.570796, 1.741233],accel_mss,speed_ms,0,blend_radius_m)
    |   movel([0.169873, -1.334543, -2.603745, -0.774101, 1.570796, 1.740669],accel_mss,speed_ms,0,blend_radius_m)
    |   movel([0.146160, -1.340657, -2.599801, -0.771931, 1.570796, 1.716956],accel_mss,speed_ms,0,blend_radius_m)
    |   movel([0.122546, -1.347144, -2.595559, -0.769685, 1.570796, 1.693343],accel_mss,speed_ms,0,blend_radius_m)
    |   movel([0.123257, -1.342070, -2.598881, -0.771437, 1.570796, 1.694053],accel_mss,speed_ms,0,blend_radius_m)
    |   movel([0.146775, -1.335675, -2.603018, -0.773695, 1.570796, 1.717571],accel_mss,speed_ms,0,blend_radius_m)
    |   movel([0.163531, -1.331456, -2.605718, -0.775216, 1.570796, 1.734328],accel_mss,speed_ms,0,blend_radius_m)
    |   movel([0.170358, -1.329852, -2.606737, -0.775800, 1.570796, 1.741154],accel_mss,speed_ms,0,blend_radius_m)
    |   movel([0.170695, -1.329903, -2.606705, -0.775781, 1.570796, 1.741491],accel_mss,speed_ms,0,blend_radius_m)
    |   movel([0.170785, -1.330115, -2.606570, -0.775704, 1.570796, 1.741581],accel_mss,speed_ms,0,blend_radius_m)
    |   movel([0.170747, -1.330725, -2.606183, -0.775481, 1.570796, 1.741543],accel_mss,speed_ms,0,blend_radius_m)
    |   movel([0.170466, -1.332197, -2.605245, -0.774947, 1.570796, 1.741263],accel_mss,speed_ms,0,blend_radius_m)
    |   speed_ms = 0.005
    |   movel([0.170466, -1.323159, -2.601032, -0.788198, 1.570796, 1.741263],accel_mss,speed_ms,0,blend_radius_m)
    |   speed_ms = 0.040
    |   movel([0.193546, -1.293118, -2.619347, -0.799924, 1.570796, 1.764342],accel_mss,speed_ms,0,blend_radius_m)
    |   speed_ms = 0.005
    |   movel([0.193546, -1.302337, -2.623694, -0.786358, 1.570796, 1.764342],accel_mss,speed_ms,0,blend_radius_m)
    |   speed_ms = 0.030
    |   movel([0.193028, -1.302847, -2.623389, -0.786153, 1.570796, 1.763825],accel_mss,speed_ms,0,blend_radius_m)
    |   movel([0.192066, -1.303300, -2.623118, -0.785971, 1.570796, 1.762862],accel_mss,speed_ms,0,blend_radius_m)
    |   movel([0.190438, -1.303811, -2.622812, -0.785767, 1.570796, 1.761235],accel_mss,speed_ms,0,blend_radius_m)
    |   movel([0.187417, -1.304576, -2.622352, -0.785461, 1.570796, 1.758213],accel_mss,speed_ms,0,blend_radius_m)
    |   movel([0.181787, -1.305968, -2.621514, -0.784907, 1.570796, 1.752583],accel_mss,speed_ms,0,blend_radius_m)
    |   movel([0.183242, -1.298721, -2.625849, -0.787819, 1.570796, 1.754038],accel_mss,speed_ms,0,blend_radius_m)
    |   movel([0.184721, -1.291389, -2.630166, -0.790834, 1.570796, 1.755517],accel_mss,speed_ms,0,blend_radius_m)
    |   movel([0.190413, -1.289951, -2.631004, -0.791434, 1.570796, 1.761209],accel_mss,speed_ms,0,blend_radius_m)
    |   movel([0.196111, -1.288729, -2.631715, -0.791945, 1.570796, 1.766907],accel_mss,speed_ms,0,blend_radius_m)
    |   movel([0.196402, -1.288787, -2.631681, -0.791921, 1.570796, 1.767198],accel_mss,speed_ms,0,blend_radius_m)
    |   movel([0.196568, -1.289056, -2.631525, -0.791808, 1.570796, 1.767365],accel_mss,speed_ms,0,blend_radius_m)
    |   movel([0.196571, -1.289422, -2.631312, -0.791655, 1.570796, 1.767367],accel_mss,speed_ms,0,blend_radius_m)
    |   movel([0.194146, -1.300833, -2.624593, -0.786963, 1.570796, 1.764942],accel_mss,speed_ms,0,blend_radius_m)
    |   movel([0.193910, -1.301581, -2.624147, -0.786662, 1.570796, 1.764706],accel_mss,speed_ms,0,blend_radius_m)
    |   movel([0.193546, -1.302337, -2.623694, -0.786358, 1.570796, 1.764342],accel_mss,speed_ms,0,blend_radius_m)
    |   movel([0.193028, -1.302847, -2.623389, -0.786153, 1.570796, 1.763825],accel_mss,speed_ms,0,blend_radius_m)
    |   movel([0.192066, -1.303300, -2.623118, -0.785971, 1.570796, 1.762862],accel_mss,speed_ms,0,blend_radius_m)
    |   movel([0.190904, -1.303665, -2.622899, -0.785825, 1.570796, 1.761700],accel_mss,speed_ms,0,blend_radius_m)
    |   speed_ms = 0.005
    |   movel([0.190904, -1.294453, -2.618557, -0.799378, 1.570796, 1.761700],accel_mss,speed_ms,0,blend_radius_m)
    |   speed_ms = 0.040
    |   movel([0.200796, -1.292139, -2.619924, -0.800326, 1.570796, 1.771592],accel_mss,speed_ms,0,blend_radius_m)
    |   speed_ms = 0.005
    |   movel([0.200796, -1.301364, -2.624276, -0.786749, 1.570796, 1.771592],accel_mss,speed_ms,0,blend_radius_m)
    |   speed_ms = 0.030
    |   movel([0.194871, -1.302770, -2.623435, -0.786184, 1.570796, 1.765668],accel_mss,speed_ms,0,blend_radius_m)
    |   movel([0.196504, -1.295565, -2.627716, -0.789109, 1.570796, 1.767300],accel_mss,speed_ms,0,blend_radius_m)
    |   movel([0.198164, -1.288274, -2.631979, -0.792136, 1.570796, 1.768960],accel_mss,speed_ms,0,blend_radius_m)
    |   movel([0.203393, -1.286864, -2.632796, -0.792729, 1.570796, 1.774189],accel_mss,speed_ms,0,blend_radius_m)
    |   movel([0.208814, -1.285584, -2.633535, -0.793270, 1.570796, 1.779610],accel_mss,speed_ms,0,blend_radius_m)
    |   movel([0.209297, -1.285563, -2.633547, -0.793279, 1.570796, 1.780093],accel_mss,speed_ms,0,blend_radius_m)
    |   movel([0.209502, -1.285668, -2.633486, -0.793234, 1.570796, 1.780299],accel_mss,speed_ms,0,blend_radius_m)
    |   movel([0.209575, -1.285888, -2.633359, -0.793141, 1.570796, 1.780371],accel_mss,speed_ms,0,blend_radius_m)
    |   movel([0.209473, -1.287177, -2.632615, -0.792597, 1.570796, 1.780269],accel_mss,speed_ms,0,blend_radius_m)
    |   movel([0.209113, -1.289278, -2.631396, -0.791715, 1.570796, 1.779909],accel_mss,speed_ms,0,blend_radius_m)
    |   movel([0.206722, -1.299983, -2.625099, -0.787307, 1.570796, 1.777519],accel_mss,speed_ms,0,blend_radius_m)
    |   movel([0.200796, -1.301364, -2.624276, -0.786749, 1.570796, 1.771592],accel_mss,speed_ms,0,blend_radius_m)
    |   movel([0.198084, -1.302004, -2.623894, -0.786491, 1.570796, 1.768880],accel_mss,speed_ms,0,blend_radius_m)
    |   speed_ms = 0.005
    |   movel([0.198084, -1.292783, -2.619544, -0.800061, 1.570796, 1.768880],accel_mss,speed_ms,0,blend_radius_m)
    |   speed_ms = 0.040
    |   movel([0.190322, -1.311159, -2.608489, -0.792741, 1.570796, 1.761118],accel_mss,speed_ms,0,blend_radius_m)
    |   speed_ms = 0.005
    |   movel([0.190322, -1.320271, -2.612756, -0.779362, 1.570796, 1.761118],accel_mss,speed_ms,0,blend_radius_m)
    |   speed_ms = 0.030
    |   movel([0.202817, -1.317404, -2.614533, -0.780452, 1.570796, 1.773614],accel_mss,speed_ms,0,blend_radius_m)
    |   movel([0.204528, -1.309750, -2.619225, -0.783415, 1.570796, 1.775324],accel_mss,speed_ms,0,blend_radius_m)
    |   movel([0.206268, -1.301999, -2.623896, -0.786493, 1.570796, 1.777065],accel_mss,speed_ms,0,blend_radius_m)
    |   movel([0.193884, -1.304905, -2.622154, -0.785330, 1.570796, 1.764681],accel_mss,speed_ms,0,blend_radius_m)
    |   movel([0.181516, -1.307921, -2.620334, -0.784134, 1.570796, 1.752313],accel_mss,speed_ms,0,blend_radius_m)
    |   movel([0.180967, -1.309116, -2.619610, -0.783664, 1.570796, 1.751764],accel_mss,speed_ms,0,blend_radius_m)
    |   movel([0.180691, -1.309881, -2.619144, -0.783363, 1.570796, 1.751488],accel_mss,speed_ms,0,blend_radius_m)
    |   movel([0.179122, -1.316813, -2.614898, -0.780678, 1.570796, 1.749918],accel_mss,speed_ms,0,blend_radius_m)
    |   movel([0.177840, -1.323251, -2.610897, -0.778241, 1.570796, 1.748636],accel_mss,speed_ms,0,blend_radius_m)
    |   movel([0.190322, -1.320271, -2.612756, -0.779362, 1.570796, 1.761118],accel_mss,speed_ms,0,blend_radius_m)
    |   movel([0.192980, -1.319652, -2.613141, -0.779597, 1.570796, 1.763776],accel_mss,speed_ms,0,blend_radius_m)
    |   speed_ms = 0.005
    |   movel([0.192980, -1.310536, -2.608871, -0.792982, 1.570796, 1.763776],accel_mss,speed_ms,0,blend_radius_m)
    |   speed_ms = 0.040
    |   movel([0.190239, -1.313969, -2.606760, -0.791660, 1.570796, 1.761036],accel_mss,speed_ms,0,blend_radius_m)
    |   speed_ms = 0.005
    |   movel([0.190239, -1.323064, -2.611014, -0.778311, 1.570796, 1.761036],accel_mss,speed_ms,0,blend_radius_m)
    |   speed_ms = 0.030
    |   movel([0.196926, -1.321501, -2.611990, -0.778898, 1.570796, 1.767722],accel_mss,speed_ms,0,blend_radius_m)
    |   movel([0.200071, -1.320689, -2.612496, -0.779204, 1.570796, 1.770868],accel_mss,speed_ms,0,blend_radius_m)
    |   movel([0.201858, -1.320104, -2.612860, -0.779425, 1.570796, 1.772655],accel_mss,speed_ms,0,blend_radius_m)
    |   movel([0.202160, -1.319902, -2.612985, -0.779502, 1.570796, 1.772957],accel_mss,speed_ms,0,blend_radius_m)
    |   movel([0.202326, -1.319609, -2.613167, -0.779613, 1.570796, 1.773123],accel_mss,speed_ms,0,blend_radius_m)
    |   movel([0.202280, -1.319364, -2.613319, -0.779706, 1.570796, 1.773076],accel_mss,speed_ms,0,blend_radius_m)
    |   movel([0.202041, -1.319283, -2.613370, -0.779736, 1.570796, 1.772837],accel_mss,speed_ms,0,blend_radius_m)
    |   movel([0.200337, -1.319483, -2.613246, -0.779661, 1.570796, 1.771133],accel_mss,speed_ms,0,blend_radius_m)
    |   movel([0.197233, -1.320087, -2.612870, -0.779431, 1.570796, 1.768030],accel_mss,speed_ms,0,blend_radius_m)
    |   movel([0.190546, -1.321607, -2.611924, -0.778858, 1.570796, 1.761342],accel_mss,speed_ms,0,blend_radius_m)
    |   movel([0.183852, -1.323208, -2.610924, -0.778257, 1.570796, 1.754649],accel_mss,speed_ms,0,blend_radius_m)
    |   movel([0.180709, -1.324059, -2.610391, -0.777939, 1.570796, 1.751505],accel_mss,speed_ms,0,blend_radius_m)
    |   movel([0.178927, -1.324670, -2.610008, -0.777711, 1.570796, 1.749724],accel_mss,speed_ms,0,blend_radius_m)
    |   movel([0.178629, -1.324875, -2.609879, -0.777635, 1.570796, 1.749426],accel_mss,speed_ms,0,blend_radius_m)
    |   movel([0.178471, -1.325166, -2.609696, -0.777527, 1.570796, 1.749267],accel_mss,speed_ms,0,blend_radius_m)
    |   movel([0.178524, -1.325406, -2.609546, -0.777438, 1.570796, 1.749321],accel_mss,speed_ms,0,blend_radius_m)
    |   movel([0.178766, -1.325480, -2.609499, -0.777410, 1.570796, 1.749563],accel_mss,speed_ms,0,blend_radius_m)
    |   movel([0.180470, -1.325251, -2.609643, -0.777495, 1.570796, 1.751266],accel_mss,speed_ms,0,blend_radius_m)
    |   movel([0.183567, -1.324610, -2.610045, -0.777733, 1.570796, 1.754363],accel_mss,speed_ms,0,blend_radius_m)
    |   movel([0.190239, -1.323064, -2.611014, -0.778311, 1.570796, 1.761036],accel_mss,speed_ms,0,blend_radius_m)
    |   movel([0.192890, -1.322440, -2.611404, -0.778545, 1.570796, 1.763687],accel_mss,speed_ms,0,blend_radius_m)
    |   speed_ms = 0.005
    |   movel([0.192890, -1.313342, -2.607147, -0.791901, 1.570796, 1.763687],accel_mss,speed_ms,0,blend_radius_m)
    |   speed_ms = 0.040
    |   movel([0.189731, -1.316404, -2.605253, -0.790732, 1.570796, 1.760527],accel_mss,speed_ms,0,blend_radius_m)
    |   speed_ms = 0.005
    |   movel([0.189731, -1.325484, -2.609496, -0.777408, 1.570796, 1.760527],accel_mss,speed_ms,0,blend_radius_m)
    |   speed_ms = 0.030
    |   movel([0.183077, -1.327021, -2.608529, -0.776840, 1.570796, 1.753873],accel_mss,speed_ms,0,blend_radius_m)
    |   movel([0.179988, -1.327657, -2.608127, -0.776605, 1.570796, 1.750785],accel_mss,speed_ms,0,blend_radius_m)
    |   movel([0.178290, -1.327884, -2.607983, -0.776521, 1.570796, 1.749086],accel_mss,speed_ms,0,blend_radius_m)
    |   movel([0.178048, -1.327810, -2.608030, -0.776549, 1.570796, 1.748844],accel_mss,speed_ms,0,blend_radius_m)
    |   movel([0.177995, -1.327571, -2.608181, -0.776637, 1.570796, 1.748791],accel_mss,speed_ms,0,blend_radius_m)
    |   movel([0.178152, -1.327282, -2.608364, -0.776743, 1.570796, 1.748949],accel_mss,speed_ms,0,blend_radius_m)
    |   movel([0.178450, -1.327078, -2.608493, -0.776819, 1.570796, 1.749246],accel_mss,speed_ms,0,blend_radius_m)
    |   movel([0.180226, -1.326470, -2.608876, -0.777043, 1.570796, 1.751022],accel_mss,speed_ms,0,blend_radius_m)
    |   movel([0.183361, -1.325624, -2.609409, -0.777357, 1.570796, 1.754157],accel_mss,speed_ms,0,blend_radius_m)
    |   movel([0.190036, -1.324033, -2.610407, -0.777949, 1.570796, 1.760832],accel_mss,speed_ms,0,blend_radius_m)
    |   movel([0.196704, -1.322523, -2.611352, -0.778514, 1.570796, 1.767501],accel_mss,speed_ms,0,blend_radius_m)
    |   movel([0.199800, -1.321923, -2.611727, -0.778739, 1.570796, 1.770596],accel_mss,speed_ms,0,blend_radius_m)
    |   movel([0.201499, -1.321724, -2.611851, -0.778814, 1.570796, 1.772295],accel_mss,speed_ms,0,blend_radius_m)
    |   movel([0.201737, -1.321805, -2.611800, -0.778783, 1.570796, 1.772534],accel_mss,speed_ms,0,blend_radius_m)
    |   movel([0.201784, -1.322050, -2.611648, -0.778691, 1.570796, 1.772580],accel_mss,speed_ms,0,blend_radius_m)
    |   movel([0.201618, -1.322341, -2.611466, -0.778582, 1.570796, 1.772415],accel_mss,speed_ms,0,blend_radius_m)
    |   movel([0.201317, -1.322543, -2.611340, -0.778506, 1.570796, 1.772114],accel_mss,speed_ms,0,blend_radius_m)
    |   movel([0.199535, -1.323124, -2.610976, -0.778288, 1.570796, 1.770331],accel_mss,speed_ms,0,blend_radius_m)
    |   movel([0.196399, -1.323932, -2.610471, -0.777986, 1.570796, 1.767195],accel_mss,speed_ms,0,blend_radius_m)
    |   movel([0.189731, -1.325484, -2.609496, -0.777408, 1.570796, 1.760527],accel_mss,speed_ms,0,blend_radius_m)
    |   movel([0.187092, -1.326090, -2.609115, -0.777184, 1.570796, 1.757888],accel_mss,speed_ms,0,blend_radius_m)
    |   speed_ms = 0.005
    |   movel([0.187092, -1.317013, -2.604875, -0.790501, 1.570796, 1.757888],accel_mss,speed_ms,0,blend_radius_m)
    |   speed_ms = 0.040
    |   movel([0.189326, -1.318346, -2.604046, -0.789997, 1.570796, 1.760122],accel_mss,speed_ms,0,blend_radius_m)
    |   speed_ms = 0.005
    |   movel([0.189326, -1.327414, -2.608281, -0.776695, 1.570796, 1.760122],accel_mss,speed_ms,0,blend_radius_m)
    |   speed_ms = 0.030
    |   movel([0.194401, -1.326222, -2.609032, -0.777135, 1.570796, 1.765197],accel_mss,speed_ms,0,blend_radius_m)
    |   movel([0.201019, -1.324513, -2.610107, -0.777770, 1.570796, 1.771815],accel_mss,speed_ms,0,blend_radius_m)
    |   movel([0.201298, -1.324238, -2.610279, -0.777872, 1.570796, 1.772094],accel_mss,speed_ms,0,blend_radius_m)
    |   movel([0.201118, -1.324066, -2.610387, -0.777936, 1.570796, 1.771914],accel_mss,speed_ms,0,blend_radius_m)
    |   movel([0.198276, -1.324573, -2.610069, -0.777747, 1.570796, 1.769072],accel_mss,speed_ms,0,blend_radius_m)
    |   movel([0.189528, -1.326450, -2.608889, -0.777051, 1.570796, 1.760325],accel_mss,speed_ms,0,blend_radius_m)
    |   movel([0.184450, -1.327663, -2.608123, -0.776603, 1.570796, 1.755246],accel_mss,speed_ms,0,blend_radius_m)
    |   movel([0.177841, -1.329453, -2.606990, -0.775946, 1.570796, 1.748637],accel_mss,speed_ms,0,blend_radius_m)
    |   movel([0.177568, -1.329728, -2.606816, -0.775845, 1.570796, 1.748364],accel_mss,speed_ms,0,blend_radius_m)
    |   movel([0.177754, -1.329893, -2.606711, -0.775785, 1.570796, 1.748550],accel_mss,speed_ms,0,blend_radius_m)
    |   movel([0.180592, -1.329343, -2.607060, -0.775986, 1.570796, 1.751388],accel_mss,speed_ms,0,blend_radius_m)
    |   movel([0.189326, -1.327414, -2.608281, -0.776695, 1.570796, 1.760122],accel_mss,speed_ms,0,blend_radius_m)
    |   movel([0.191965, -1.326793, -2.608673, -0.776924, 1.570796, 1.762761],accel_mss,speed_ms,0,blend_radius_m)
    |   speed_ms = 0.005
    |   movel([0.191965, -1.317721, -2.604435, -0.790233, 1.570796, 1.762761],accel_mss,speed_ms,0,blend_radius_m)
    |   speed_ms = 0.040
    |   movel([0.192708, -1.351839, -2.582429, -0.778122, 1.570796, 1.763505],accel_mss,speed_ms,0,blend_radius_m)
    |   speed_ms = 0.005
    |   movel([0.192708, -1.360690, -2.586515, -0.765184, 1.570796, 1.763505],accel_mss,speed_ms,0,blend_radius_m)
    |   speed_ms = 0.030
    |   movel([0.192968, -1.360550, -2.586610, -0.765229, 1.570796, 1.763764],accel_mss,speed_ms,0,blend_radius_m)
    |   movel([0.193123, -1.360312, -2.586771, -0.765306, 1.570796, 1.763920],accel_mss,speed_ms,0,blend_radius_m)
    |   movel([0.193962, -1.357104, -2.588934, -0.766351, 1.570796, 1.764759],accel_mss,speed_ms,0,blend_radius_m)
    |   movel([0.197033, -1.343588, -2.597892, -0.770910, 1.570796, 1.767830],accel_mss,speed_ms,0,blend_radius_m)
    |   movel([0.200872, -1.326160, -2.609071, -0.777158, 1.570796, 1.771668],accel_mss,speed_ms,0,blend_radius_m)
    |   movel([0.188606, -1.329059, -2.607240, -0.776090, 1.570796, 1.759402],accel_mss,speed_ms,0,blend_radius_m)
    |   movel([0.176356, -1.332067, -2.605328, -0.774994, 1.570796, 1.747152],accel_mss,speed_ms,0,blend_radius_m)
    |   movel([0.169216, -1.367579, -2.581817, -0.762993, 1.570796, 1.740012],accel_mss,speed_ms,0,blend_radius_m)
    |   movel([0.170610, -1.367259, -2.582036, -0.763094, 1.570796, 1.741407],accel_mss,speed_ms,0,blend_radius_m)
    |   movel([0.174533, -1.366122, -2.582816, -0.763451, 1.570796, 1.745329],accel_mss,speed_ms,0,blend_radius_m)
    |   movel([0.178080, -1.365054, -2.583547, -0.763789, 1.570796, 1.748877],accel_mss,speed_ms,0,blend_radius_m)
    |   movel([0.192708, -1.360690, -2.586515, -0.765184, 1.570796, 1.763505],accel_mss,speed_ms,0,blend_radius_m)
    |   movel([0.192968, -1.360550, -2.586610, -0.765229, 1.570796, 1.763764],accel_mss,speed_ms,0,blend_radius_m)
    |   movel([0.193123, -1.360312, -2.586771, -0.765306, 1.570796, 1.763920],accel_mss,speed_ms,0,blend_radius_m)
    |   movel([0.193605, -1.358473, -2.588013, -0.765903, 1.570796, 1.764402],accel_mss,speed_ms,0,blend_radius_m)
    |   speed_ms = 0.005
    |   movel([0.193605, -1.349606, -2.583917, -0.778866, 1.570796, 1.764402],accel_mss,speed_ms,0,blend_radius_m)
    |   speed_ms = 0.040
    |   movel([0.190579, -1.355040, -2.580282, -0.777066, 1.570796, 1.761375],accel_mss,speed_ms,0,blend_radius_m)
    |   speed_ms = 0.005
    |   movel([0.190579, -1.363870, -2.584354, -0.764164, 1.570796, 1.761375],accel_mss,speed_ms,0,blend_radius_m)
    |   speed_ms = 0.030
    |   movel([0.191428, -1.363571, -2.584558, -0.764260, 1.570796, 1.762224],accel_mss,speed_ms,0,blend_radius_m)
    |   movel([0.192707, -1.362964, -2.584971, -0.764453, 1.570796, 1.763504],accel_mss,speed_ms,0,blend_radius_m)
    |   movel([0.192847, -1.362632, -2.585197, -0.764560, 1.570796, 1.763643],accel_mss,speed_ms,0,blend_radius_m)
    |   movel([0.192313, -1.362524, -2.585271, -0.764594, 1.570796, 1.763109],accel_mss,speed_ms,0,blend_radius_m)
    |   movel([0.189361, -1.363311, -2.584736, -0.764343, 1.570796, 1.760157],accel_mss,speed_ms,0,blend_radius_m)
    |   movel([0.167815, -1.370067, -2.580103, -0.762219, 1.570796, 1.738611],accel_mss,speed_ms,0,blend_radius_m)
    |   movel([0.167375, -1.370335, -2.579918, -0.762136, 1.570796, 1.738171],accel_mss,speed_ms,0,blend_radius_m)
    |   movel([0.167255, -1.370596, -2.579738, -0.762055, 1.570796, 1.738052],accel_mss,speed_ms,0,blend_radius_m)
    |   movel([0.167425, -1.370729, -2.579646, -0.762014, 1.570796, 1.738221],accel_mss,speed_ms,0,blend_radius_m)
    |   movel([0.168786, -1.370559, -2.579764, -0.762067, 1.570796, 1.739583],accel_mss,speed_ms,0,blend_radius_m)
    |   movel([0.171912, -1.369702, -2.580355, -0.762332, 1.570796, 1.742708],accel_mss,speed_ms,0,blend_radius_m)
    |   movel([0.190579, -1.363870, -2.584354, -0.764164, 1.570796, 1.761375],accel_mss,speed_ms,0,blend_radius_m)
    |   movel([0.191428, -1.363571, -2.584558, -0.764260, 1.570796, 1.762224],accel_mss,speed_ms,0,blend_radius_m)
    |   movel([0.192707, -1.362964, -2.584971, -0.764453, 1.570796, 1.763504],accel_mss,speed_ms,0,blend_radius_m)
    |   movel([0.192847, -1.362632, -2.585197, -0.764560, 1.570796, 1.763643],accel_mss,speed_ms,0,blend_radius_m)
    |   speed_ms = 0.005
    |   movel([0.192847, -1.353794, -2.581120, -0.777476, 1.570796, 1.763643],accel_mss,speed_ms,0,blend_radius_m)
    |   speed_ms = 0.040
    |   movel([0.192479, -1.356286, -2.579443, -0.776660, 1.570796, 1.763275],accel_mss,speed_ms,0,blend_radius_m)
    |   speed_ms = 0.005
    |   movel([0.192479, -1.365107, -2.583510, -0.763772, 1.570796, 1.763275],accel_mss,speed_ms,0,blend_radius_m)
    |   speed_ms = 0.030
    |   movel([0.192847, -1.364872, -2.583671, -0.763846, 1.570796, 1.763643],accel_mss,speed_ms,0,blend_radius_m)
    |   movel([0.192945, -1.364549, -2.583891, -0.763949, 1.570796, 1.763742],accel_mss,speed_ms,0,blend_radius_m)
    |   movel([0.192671, -1.364293, -2.584066, -0.764030, 1.570796, 1.763467],accel_mss,speed_ms,0,blend_radius_m)
    |   movel([0.192176, -1.364280, -2.584075, -0.764034, 1.570796, 1.762972],accel_mss,speed_ms,0,blend_radius_m)
    |   movel([0.190050, -1.364826, -2.583703, -0.763861, 1.570796, 1.760846],accel_mss,speed_ms,0,blend_radius_m)
    |   movel([0.167353, -1.371984, -2.578777, -0.761628, 1.570796, 1.738149],accel_mss,speed_ms,0,blend_radius_m)
    |   movel([0.166931, -1.372234, -2.578604, -0.761551, 1.570796, 1.737728],accel_mss,speed_ms,0,blend_radius_m)
    |   movel([0.166803, -1.372522, -2.578404, -0.761463, 1.570796, 1.737599],accel_mss,speed_ms,0,blend_radius_m)
    |   movel([0.167006, -1.372651, -2.578314, -0.761423, 1.570796, 1.737802],accel_mss,speed_ms,0,blend_radius_m)
    |   movel([0.168962, -1.372304, -2.578555, -0.761530, 1.570796, 1.739758],accel_mss,speed_ms,0,blend_radius_m)
    |   movel([0.172891, -1.371208, -2.579315, -0.761867, 1.570796, 1.743688],accel_mss,speed_ms,0,blend_radius_m)
    |   movel([0.192479, -1.365107, -2.583510, -0.763772, 1.570796, 1.763275],accel_mss,speed_ms,0,blend_radius_m)
    |   movel([0.192847, -1.364872, -2.583671, -0.763846, 1.570796, 1.763643],accel_mss,speed_ms,0,blend_radius_m)
    |   movel([0.192945, -1.364549, -2.583891, -0.763949, 1.570796, 1.763742],accel_mss,speed_ms,0,blend_radius_m)
    |   movel([0.192671, -1.364293, -2.584066, -0.764030, 1.570796, 1.763467],accel_mss,speed_ms,0,blend_radius_m)
    |   movel([0.192176, -1.364280, -2.584075, -0.764034, 1.570796, 1.762972],accel_mss,speed_ms,0,blend_radius_m)
    |   movel([0.191422, -1.364473, -2.583943, -0.763973, 1.570796, 1.762218],accel_mss,speed_ms,0,blend_radius_m)
    |   speed_ms = 0.005
    |   movel([0.191422, -1.355647, -2.579874, -0.776868, 1.570796, 1.762218],accel_mss,speed_ms,0,blend_radius_m)
    |   speed_ms = 0.040
    |   movel([0.189787, -1.364153, -2.574095, -0.774141, 1.570796, 1.760584],accel_mss,speed_ms,0,blend_radius_m)
    |   speed_ms = 0.005
    |   movel([0.189787, -1.372920, -2.578128, -0.761341, 1.570796, 1.760584],accel_mss,speed_ms,0,blend_radius_m)
    |   speed_ms = 0.030
    |   movel([0.190802, -1.371736, -2.578949, -0.761704, 1.570796, 1.761598],accel_mss,speed_ms,0,blend_radius_m)
    |   movel([0.191525, -1.370690, -2.579673, -0.762026, 1.570796, 1.762322],accel_mss,speed_ms,0,blend_radius_m)
    |   movel([0.192069, -1.369599, -2.580426, -0.762364, 1.570796, 1.762865],accel_mss,speed_ms,0,blend_radius_m)
    |   movel([0.192539, -1.368274, -2.581339, -0.762776, 1.570796, 1.763335],accel_mss,speed_ms,0,blend_radius_m)
    |   movel([0.192725, -1.367437, -2.581914, -0.763038, 1.570796, 1.763521],accel_mss,speed_ms,0,blend_radius_m)
    |   movel([0.192760, -1.366639, -2.582462, -0.763288, 1.570796, 1.763557],accel_mss,speed_ms,0,blend_radius_m)
    |   movel([0.192564, -1.366270, -2.582714, -0.763404, 1.570796, 1.763360],accel_mss,speed_ms,0,blend_radius_m)
    |   movel([0.192094, -1.366180, -2.582776, -0.763433, 1.570796, 1.762890],accel_mss,speed_ms,0,blend_radius_m)
    |   movel([0.190038, -1.366628, -2.582469, -0.763292, 1.570796, 1.760834],accel_mss,speed_ms,0,blend_radius_m)
    |   movel([0.178831, -1.370102, -2.580079, -0.762208, 1.570796, 1.749628],accel_mss,speed_ms,0,blend_radius_m)
    |   movel([0.166819, -1.373936, -2.577422, -0.761032, 1.570796, 1.737615],accel_mss,speed_ms,0,blend_radius_m)
    |   movel([0.165845, -1.378365, -2.574325, -0.759699, 1.570796, 1.736641],accel_mss,speed_ms,0,blend_radius_m)
    |   movel([0.165504, -1.380078, -2.573120, -0.759191, 1.570796, 1.736300],accel_mss,speed_ms,0,blend_radius_m)
    |   movel([0.165157, -1.382777, -2.571213, -0.758399, 1.570796, 1.735953],accel_mss,speed_ms,0,blend_radius_m)
    |   movel([0.165274, -1.383075, -2.571001, -0.758312, 1.570796, 1.736070],accel_mss,speed_ms,0,blend_radius_m)
    |   movel([0.165728, -1.383281, -2.570855, -0.758252, 1.570796, 1.736525],accel_mss,speed_ms,0,blend_radius_m)
    |   movel([0.166306, -1.383296, -2.570845, -0.758248, 1.570796, 1.737103],accel_mss,speed_ms,0,blend_radius_m)
    |   movel([0.169378, -1.382785, -2.571207, -0.758397, 1.570796, 1.740174],accel_mss,speed_ms,0,blend_radius_m)
    |   movel([0.172884, -1.381985, -2.571773, -0.758630, 1.570796, 1.743681],accel_mss,speed_ms,0,blend_radius_m)
    |   movel([0.176221, -1.380973, -2.572489, -0.758927, 1.570796, 1.747017],accel_mss,speed_ms,0,blend_radius_m)
    |   movel([0.178197, -1.380232, -2.573011, -0.759145, 1.570796, 1.748994],accel_mss,speed_ms,0,blend_radius_m)
    |   movel([0.180168, -1.379381, -2.573611, -0.759397, 1.570796, 1.750964],accel_mss,speed_ms,0,blend_radius_m)
    |   movel([0.182082, -1.378434, -2.574276, -0.759678, 1.570796, 1.752878],accel_mss,speed_ms,0,blend_radius_m)
    |   movel([0.183972, -1.377377, -2.575018, -0.759994, 1.570796, 1.754769],accel_mss,speed_ms,0,blend_radius_m)
    |   movel([0.185660, -1.376317, -2.575761, -0.760312, 1.570796, 1.756456],accel_mss,speed_ms,0,blend_radius_m)
    |   movel([0.187300, -1.375157, -2.576571, -0.760661, 1.570796, 1.758096],accel_mss,speed_ms,0,blend_radius_m)
    |   movel([0.188599, -1.374092, -2.577313, -0.760984, 1.570796, 1.759395],accel_mss,speed_ms,0,blend_radius_m)
    |   movel([0.189787, -1.372920, -2.578128, -0.761341, 1.570796, 1.760584],accel_mss,speed_ms,0,blend_radius_m)
    |   movel([0.190802, -1.371736, -2.578949, -0.761704, 1.570796, 1.761598],accel_mss,speed_ms,0,blend_radius_m)
    |   movel([0.191494, -1.370736, -2.579641, -0.762012, 1.570796, 1.762290],accel_mss,speed_ms,0,blend_radius_m)
    |   speed_ms = 0.005
    |   movel([0.191494, -1.361953, -2.575599, -0.774837, 1.570796, 1.762290],accel_mss,speed_ms,0,blend_radius_m)
    |   speed_ms = 0.040
    |   movel([0.160550, -1.340565, -2.589874, -0.781949, 1.570796, 1.731347],accel_mss,speed_ms,0,blend_radius_m)
    |   speed_ms = 0.005
    |   movel([0.160550, -1.349491, -2.594010, -0.768887, 1.570796, 1.731347],accel_mss,speed_ms,0,blend_radius_m)
    |   speed_ms = 0.030
    |   movel([0.159643, -1.348682, -2.594545, -0.769162, 1.570796, 1.730439],accel_mss,speed_ms,0,blend_radius_m)
    |   movel([0.158990, -1.348358, -2.594759, -0.769272, 1.570796, 1.729786],accel_mss,speed_ms,0,blend_radius_m)
    |   movel([0.157463, -1.347924, -2.595046, -0.769419, 1.570796, 1.728260],accel_mss,speed_ms,0,blend_radius_m)
    |   movel([0.157062, -1.347597, -2.595261, -0.769531, 1.570796, 1.727858],accel_mss,speed_ms,0,blend_radius_m)
    |   movel([0.156944, -1.347046, -2.595624, -0.769719, 1.570796, 1.727740],accel_mss,speed_ms,0,blend_radius_m)
    |   movel([0.157070, -1.345995, -2.596315, -0.770079, 1.570796, 1.727867],accel_mss,speed_ms,0,blend_radius_m)
    |   movel([0.157187, -1.345124, -2.596886, -0.770379, 1.570796, 1.727983],accel_mss,speed_ms,0,blend_radius_m)
    |   movel([0.157146, -1.344601, -2.597229, -0.770559, 1.570796, 1.727942],accel_mss,speed_ms,0,blend_radius_m)
    |   movel([0.156957, -1.344351, -2.597393, -0.770646, 1.570796, 1.727753],accel_mss,speed_ms,0,blend_radius_m)
    |   movel([0.156621, -1.344323, -2.597411, -0.770655, 1.570796, 1.727418],accel_mss,speed_ms,0,blend_radius_m)
    |   movel([0.156238, -1.344542, -2.597268, -0.770580, 1.570796, 1.727034],accel_mss,speed_ms,0,blend_radius_m)
    |   movel([0.155934, -1.344940, -2.597007, -0.770442, 1.570796, 1.726731],accel_mss,speed_ms,0,blend_radius_m)
    |   movel([0.155689, -1.345590, -2.596581, -0.770218, 1.570796, 1.726485],accel_mss,speed_ms,0,blend_radius_m)
    |   movel([0.155476, -1.346608, -2.595912, -0.769869, 1.570796, 1.726272],accel_mss,speed_ms,0,blend_radius_m)
    |   movel([0.155259, -1.347650, -2.595226, -0.769513, 1.570796, 1.726055],accel_mss,speed_ms,0,blend_radius_m)
    |   movel([0.155013, -1.348288, -2.594805, -0.769295, 1.570796, 1.725810],accel_mss,speed_ms,0,blend_radius_m)
    |   movel([0.154704, -1.348675, -2.594550, -0.769164, 1.570796, 1.725500],accel_mss,speed_ms,0,blend_radius_m)
    |   movel([0.154297, -1.348894, -2.594405, -0.769090, 1.570796, 1.725093],accel_mss,speed_ms,0,blend_radius_m)
    |   movel([0.153869, -1.349083, -2.594280, -0.769026, 1.570796, 1.724665],accel_mss,speed_ms,0,blend_radius_m)
    |   movel([0.153208, -1.349547, -2.593974, -0.768869, 1.570796, 1.724004],accel_mss,speed_ms,0,blend_radius_m)
    |   movel([0.151741, -1.350825, -2.593127, -0.768437, 1.570796, 1.722537],accel_mss,speed_ms,0,blend_radius_m)
    |   movel([0.150833, -1.351808, -2.592474, -0.768107, 1.570796, 1.721629],accel_mss,speed_ms,0,blend_radius_m)
    |   movel([0.150269, -1.352626, -2.591930, -0.767833, 1.570796, 1.721066],accel_mss,speed_ms,0,blend_radius_m)
    |   movel([0.149909, -1.353502, -2.591346, -0.767541, 1.570796, 1.720705],accel_mss,speed_ms,0,blend_radius_m)
    |   movel([0.149643, -1.354677, -2.590561, -0.767151, 1.570796, 1.720439],accel_mss,speed_ms,0,blend_radius_m)
    |   movel([0.149517, -1.355816, -2.589799, -0.766774, 1.570796, 1.720313],accel_mss,speed_ms,0,blend_radius_m)
    |   movel([0.149599, -1.356577, -2.589288, -0.766524, 1.570796, 1.720395],accel_mss,speed_ms,0,blend_radius_m)
    |   movel([0.149920, -1.357168, -2.588891, -0.766330, 1.570796, 1.720717],accel_mss,speed_ms,0,blend_radius_m)
    |   movel([0.151100, -1.358111, -2.588257, -0.766022, 1.570796, 1.721896],accel_mss,speed_ms,0,blend_radius_m)
    |   movel([0.151686, -1.358377, -2.588077, -0.765935, 1.570796, 1.722482],accel_mss,speed_ms,0,blend_radius_m)
    |   movel([0.152234, -1.358535, -2.587971, -0.765883, 1.570796, 1.723030],accel_mss,speed_ms,0,blend_radius_m)
    |   movel([0.152628, -1.358519, -2.587982, -0.765888, 1.570796, 1.723424],accel_mss,speed_ms,0,blend_radius_m)
    |   movel([0.152988, -1.358545, -2.587964, -0.765880, 1.570796, 1.723784],accel_mss,speed_ms,0,blend_radius_m)
    |   movel([0.153183, -1.358802, -2.587791, -0.765796, 1.570796, 1.723979],accel_mss,speed_ms,0,blend_radius_m)
    |   movel([0.153218, -1.359361, -2.587413, -0.765614, 1.570796, 1.724014],accel_mss,speed_ms,0,blend_radius_m)
    |   movel([0.153078, -1.360365, -2.586735, -0.765289, 1.570796, 1.723874],accel_mss,speed_ms,0,blend_radius_m)
    |   movel([0.152919, -1.361480, -2.585979, -0.764929, 1.570796, 1.723715],accel_mss,speed_ms,0,blend_radius_m)
    |   movel([0.152972, -1.361990, -2.585634, -0.764766, 1.570796, 1.723768],accel_mss,speed_ms,0,blend_radius_m)
    |   movel([0.153233, -1.362186, -2.585500, -0.764703, 1.570796, 1.724029],accel_mss,speed_ms,0,blend_radius_m)
    |   movel([0.153742, -1.362155, -2.585521, -0.764713, 1.570796, 1.724538],accel_mss,speed_ms,0,blend_radius_m)
    |   movel([0.154285, -1.361931, -2.585673, -0.764784, 1.570796, 1.725082],accel_mss,speed_ms,0,blend_radius_m)
    |   movel([0.154637, -1.361592, -2.585903, -0.764893, 1.570796, 1.725433],accel_mss,speed_ms,0,blend_radius_m)
    |   movel([0.154881, -1.361018, -2.586292, -0.765078, 1.570796, 1.725678],accel_mss,speed_ms,0,blend_radius_m)
    |   movel([0.155108, -1.359920, -2.587036, -0.765433, 1.570796, 1.725904],accel_mss,speed_ms,0,blend_radius_m)
    |   movel([0.155358, -1.358778, -2.587807, -0.765804, 1.570796, 1.726154],accel_mss,speed_ms,0,blend_radius_m)
    |   movel([0.155657, -1.358119, -2.588251, -0.766019, 1.570796, 1.726453],accel_mss,speed_ms,0,blend_radius_m)
    |   movel([0.156141, -1.357608, -2.588595, -0.766186, 1.570796, 1.726937],accel_mss,speed_ms,0,blend_radius_m)
    |   movel([0.156989, -1.357048, -2.588972, -0.766369, 1.570796, 1.727785],accel_mss,speed_ms,0,blend_radius_m)
    |   movel([0.158031, -1.356333, -2.589452, -0.766604, 1.570796, 1.728828],accel_mss,speed_ms,0,blend_radius_m)
    |   movel([0.158955, -1.355467, -2.590032, -0.766889, 1.570796, 1.729752],accel_mss,speed_ms,0,blend_radius_m)
    |   movel([0.159760, -1.354452, -2.590711, -0.767225, 1.570796, 1.730557],accel_mss,speed_ms,0,blend_radius_m)
    |   movel([0.160375, -1.353386, -2.591423, -0.767580, 1.570796, 1.731171],accel_mss,speed_ms,0,blend_radius_m)
    |   movel([0.160781, -1.352296, -2.592150, -0.767943, 1.570796, 1.731577],accel_mss,speed_ms,0,blend_radius_m)
    |   movel([0.160955, -1.351241, -2.592851, -0.768297, 1.570796, 1.731751],accel_mss,speed_ms,0,blend_radius_m)
    |   movel([0.160879, -1.350301, -2.593475, -0.768614, 1.570796, 1.731676],accel_mss,speed_ms,0,blend_radius_m)
    |   movel([0.160550, -1.349491, -2.594010, -0.768887, 1.570796, 1.731347],accel_mss,speed_ms,0,blend_radius_m)
    |   movel([0.159643, -1.348682, -2.594545, -0.769162, 1.570796, 1.730439],accel_mss,speed_ms,0,blend_radius_m)
    |   movel([0.158990, -1.348358, -2.594759, -0.769272, 1.570796, 1.729786],accel_mss,speed_ms,0,blend_radius_m)
    |   speed_ms = 0.005
    |   movel([0.158990, -1.339425, -2.590618, -0.782346, 1.570796, 1.729786],accel_mss,speed_ms,0,blend_radius_m)
    |   speed_ms = 0.040
    |   movel([0.142079, -1.345416, -2.586692, -0.780281, 1.570796, 1.712875],accel_mss,speed_ms,0,blend_radius_m)
    |   speed_ms = 0.005
    |   movel([0.142079, -1.354310, -2.590807, -0.767272, 1.570796, 1.712875],accel_mss,speed_ms,0,blend_radius_m)
    |   speed_ms = 0.030
    |   movel([0.142414, -1.355424, -2.590062, -0.766904, 1.570796, 1.713211],accel_mss,speed_ms,0,blend_radius_m)
    |   movel([0.142434, -1.356228, -2.589522, -0.766638, 1.570796, 1.713231],accel_mss,speed_ms,0,blend_radius_m)
    |   movel([0.142151, -1.357116, -2.588926, -0.766347, 1.570796, 1.712947],accel_mss,speed_ms,0,blend_radius_m)
    |   movel([0.141422, -1.358517, -2.587983, -0.765889, 1.570796, 1.712218],accel_mss,speed_ms,0,blend_radius_m)
    |   movel([0.140871, -1.359349, -2.587421, -0.765618, 1.570796, 1.711667],accel_mss,speed_ms,0,blend_radius_m)
    |   movel([0.140186, -1.360139, -2.586888, -0.765362, 1.570796, 1.710982],accel_mss,speed_ms,0,blend_radius_m)
    |   movel([0.139387, -1.360864, -2.586397, -0.765128, 1.570796, 1.710184],accel_mss,speed_ms,0,blend_radius_m)
    |   movel([0.138495, -1.361505, -2.585963, -0.764921, 1.570796, 1.709291],accel_mss,speed_ms,0,blend_radius_m)
    |   movel([0.137408, -1.362254, -2.585454, -0.764681, 1.570796, 1.708205],accel_mss,speed_ms,0,blend_radius_m)
    |   movel([0.136841, -1.362817, -2.585071, -0.764500, 1.570796, 1.707637],accel_mss,speed_ms,0,blend_radius_m)
    |   movel([0.136514, -1.363454, -2.584638, -0.764297, 1.570796, 1.707311],accel_mss,speed_ms,0,blend_radius_m)
    |   movel([0.136296, -1.364450, -2.583959, -0.763980, 1.570796, 1.707092],accel_mss,speed_ms,0,blend_radius_m)
    |   movel([0.136131, -1.365261, -2.583405, -0.763723, 1.570796, 1.706927],accel_mss,speed_ms,0,blend_radius_m)
    |   movel([0.135914, -1.365809, -2.583030, -0.763550, 1.570796, 1.706710],accel_mss,speed_ms,0,blend_radius_m)
    |   movel([0.135631, -1.366160, -2.582790, -0.763439, 1.570796, 1.706427],accel_mss,speed_ms,0,blend_radius_m)
    |   movel([0.135269, -1.366356, -2.582656, -0.763377, 1.570796, 1.706065],accel_mss,speed_ms,0,blend_radius_m)
    |   movel([0.134940, -1.366337, -2.582668, -0.763383, 1.570796, 1.705737],accel_mss,speed_ms,0,blend_radius_m)
    |   movel([0.134746, -1.366110, -2.582824, -0.763455, 1.570796, 1.705543],accel_mss,speed_ms,0,blend_radius_m)
    |   movel([0.134688, -1.365633, -2.583150, -0.763605, 1.570796, 1.705484],accel_mss,speed_ms,0,blend_radius_m)
    |   movel([0.134770, -1.364844, -2.583690, -0.763855, 1.570796, 1.705567],accel_mss,speed_ms,0,blend_radius_m)
    |   movel([0.134855, -1.363883, -2.584346, -0.764160, 1.570796, 1.705651],accel_mss,speed_ms,0,blend_radius_m)
    |   movel([0.134706, -1.363370, -2.584695, -0.764324, 1.570796, 1.705503],accel_mss,speed_ms,0,blend_radius_m)
    |   movel([0.134273, -1.363066, -2.584902, -0.764421, 1.570796, 1.705070],accel_mss,speed_ms,0,blend_radius_m)
    |   movel([0.133339, -1.362841, -2.585055, -0.764493, 1.570796, 1.704135],accel_mss,speed_ms,0,blend_radius_m)
    |   movel([0.132197, -1.362438, -2.585329, -0.764622, 1.570796, 1.702994],accel_mss,speed_ms,0,blend_radius_m)
    |   movel([0.131369, -1.361690, -2.585837, -0.764862, 1.570796, 1.702165],accel_mss,speed_ms,0,blend_radius_m)
    |   movel([0.130923, -1.360653, -2.586540, -0.765196, 1.570796, 1.701719],accel_mss,speed_ms,0,blend_radius_m)
    |   movel([0.130893, -1.359402, -2.587386, -0.765601, 1.570796, 1.701690],accel_mss,speed_ms,0,blend_radius_m)
    |   movel([0.131287, -1.358022, -2.588317, -0.766051, 1.570796, 1.702083],accel_mss,speed_ms,0,blend_radius_m)
    |   movel([0.132070, -1.356631, -2.589252, -0.766506, 1.570796, 1.702866],accel_mss,speed_ms,0,blend_radius_m)
    |   movel([0.133193, -1.355318, -2.590133, -0.766939, 1.570796, 1.703990],accel_mss,speed_ms,0,blend_radius_m)
    |   movel([0.134560, -1.354192, -2.590886, -0.767312, 1.570796, 1.705357],accel_mss,speed_ms,0,blend_radius_m)
    |   movel([0.135719, -1.353341, -2.591453, -0.767594, 1.570796, 1.706516],accel_mss,speed_ms,0,blend_radius_m)
    |   movel([0.136327, -1.352721, -2.591866, -0.767801, 1.570796, 1.707123],accel_mss,speed_ms,0,blend_radius_m)
    |   movel([0.136673, -1.352054, -2.592311, -0.768024, 1.570796, 1.707469],accel_mss,speed_ms,0,blend_radius_m)
    |   movel([0.136900, -1.351055, -2.592974, -0.768360, 1.570796, 1.707696],accel_mss,speed_ms,0,blend_radius_m)
    |   movel([0.137068, -1.350243, -2.593512, -0.768633, 1.570796, 1.707865],accel_mss,speed_ms,0,blend_radius_m)
    |   movel([0.137289, -1.349688, -2.593880, -0.768821, 1.570796, 1.708085],accel_mss,speed_ms,0,blend_radius_m)
    |   movel([0.137578, -1.349332, -2.594116, -0.768941, 1.570796, 1.708374],accel_mss,speed_ms,0,blend_radius_m)
    |   movel([0.137947, -1.349129, -2.594250, -0.769010, 1.570796, 1.708743],accel_mss,speed_ms,0,blend_radius_m)
    |   movel([0.138282, -1.349146, -2.594239, -0.769004, 1.570796, 1.709078],accel_mss,speed_ms,0,blend_radius_m)
    |   movel([0.138479, -1.349379, -2.594085, -0.768925, 1.570796, 1.709275],accel_mss,speed_ms,0,blend_radius_m)
    |   movel([0.138536, -1.349867, -2.593761, -0.768760, 1.570796, 1.709332],accel_mss,speed_ms,0,blend_radius_m)
    |   movel([0.138449, -1.350675, -2.593226, -0.768487, 1.570796, 1.709245],accel_mss,speed_ms,0,blend_radius_m)
    |   movel([0.138359, -1.351656, -2.592575, -0.768158, 1.570796, 1.709155],accel_mss,speed_ms,0,blend_radius_m)
    |   movel([0.138507, -1.352179, -2.592227, -0.767982, 1.570796, 1.709303],accel_mss,speed_ms,0,blend_radius_m)
    |   movel([0.138943, -1.352488, -2.592022, -0.767879, 1.570796, 1.709739],accel_mss,speed_ms,0,blend_radius_m)
    |   movel([0.139883, -1.352718, -2.591868, -0.767802, 1.570796, 1.710679],accel_mss,speed_ms,0,blend_radius_m)
    |   movel([0.140618, -1.352928, -2.591729, -0.767732, 1.570796, 1.711414],accel_mss,speed_ms,0,blend_radius_m)
    |   movel([0.141262, -1.353285, -2.591491, -0.767613, 1.570796, 1.712058],accel_mss,speed_ms,0,blend_radius_m)
    |   movel([0.141761, -1.353758, -2.591176, -0.767456, 1.570796, 1.712557],accel_mss,speed_ms,0,blend_radius_m)
    |   movel([0.142079, -1.354310, -2.590807, -0.767272, 1.570796, 1.712875],accel_mss,speed_ms,0,blend_radius_m)
    |   movel([0.142414, -1.355424, -2.590062, -0.766904, 1.570796, 1.713211],accel_mss,speed_ms,0,blend_radius_m)
    |   movel([0.142434, -1.356228, -2.589522, -0.766638, 1.570796, 1.713231],accel_mss,speed_ms,0,blend_radius_m)
    |   speed_ms = 0.005
    |   movel([0.142434, -1.347347, -2.585416, -0.779626, 1.570796, 1.713231],accel_mss,speed_ms,0,blend_radius_m)
    |   speed_ms = 0.040
    |   movel([0.153851, -1.354795, -2.580447, -0.777147, 1.570796, 1.724647],accel_mss,speed_ms,0,blend_radius_m)
    |   speed_ms = 0.005
    |   movel([0.153851, -1.363626, -2.584521, -0.764242, 1.570796, 1.724647],accel_mss,speed_ms,0,blend_radius_m)
    |   speed_ms = 0.030
    |   movel([0.153343, -1.363665, -2.584494, -0.764230, 1.570796, 1.724139],accel_mss,speed_ms,0,blend_radius_m)
    |   movel([0.145446, -1.365581, -2.583186, -0.763622, 1.570796, 1.716242],accel_mss,speed_ms,0,blend_radius_m)
    |   movel([0.099137, -1.378020, -2.574568, -0.759802, 1.570796, 1.669934],accel_mss,speed_ms,0,blend_radius_m)
    |   movel([0.097952, -1.388375, -2.567224, -0.756791, 1.570796, 1.668749],accel_mss,speed_ms,0,blend_radius_m)
    |   movel([0.096796, -1.398572, -2.559840, -0.753977, 1.570796, 1.667592],accel_mss,speed_ms,0,blend_radius_m)
    |   movel([0.122595, -1.391852, -2.564723, -0.755814, 1.570796, 1.693391],accel_mss,speed_ms,0,blend_radius_m)
    |   movel([0.148775, -1.385385, -2.569360, -0.757644, 1.570796, 1.719571],accel_mss,speed_ms,0,blend_radius_m)
    |   movel([0.149665, -1.385085, -2.569574, -0.757731, 1.570796, 1.720461],accel_mss,speed_ms,0,blend_radius_m)
    |   movel([0.150820, -1.384582, -2.569932, -0.757876, 1.570796, 1.721617],accel_mss,speed_ms,0,blend_radius_m)
    |   movel([0.152612, -1.374219, -2.577224, -0.760945, 1.570796, 1.723408],accel_mss,speed_ms,0,blend_radius_m)
    |   movel([0.153921, -1.365951, -2.582933, -0.763505, 1.570796, 1.724717],accel_mss,speed_ms,0,blend_radius_m)
    |   movel([0.154117, -1.363937, -2.584308, -0.764143, 1.570796, 1.724914],accel_mss,speed_ms,0,blend_radius_m)
    |   movel([0.154055, -1.363723, -2.584454, -0.764211, 1.570796, 1.724851],accel_mss,speed_ms,0,blend_radius_m)
    |   movel([0.153851, -1.363626, -2.584521, -0.764242, 1.570796, 1.724647],accel_mss,speed_ms,0,blend_radius_m)
    |   movel([0.153343, -1.363665, -2.584494, -0.764230, 1.570796, 1.724139],accel_mss,speed_ms,0,blend_radius_m)
    |   movel([0.151339, -1.364148, -2.584165, -0.764076, 1.570796, 1.722135],accel_mss,speed_ms,0,blend_radius_m)
    |   speed_ms = 0.005
    |   movel([0.151339, -1.355321, -2.580094, -0.776975, 1.570796, 1.722135],accel_mss,speed_ms,0,blend_radius_m)
    |   speed_ms = 0.040
    |   movel([0.123568, -1.384726, -2.559697, -0.767965, 1.570796, 1.694365],accel_mss,speed_ms,0,blend_radius_m)
    |   speed_ms = 0.005
    |   movel([0.123568, -1.393350, -2.563640, -0.755399, 1.570796, 1.694365],accel_mss,speed_ms,0,blend_radius_m)
    |   speed_ms = 0.030
    |   movel([0.084125, -1.403925, -2.555903, -0.752562, 1.570796, 1.654922],accel_mss,speed_ms,0,blend_radius_m)
    |   movel([0.088158, -1.363791, -2.584408, -0.764190, 1.570796, 1.658955],accel_mss,speed_ms,0,blend_radius_m)
    |   movel([0.092605, -1.321074, -2.612256, -0.779059, 1.570796, 1.663401],accel_mss,speed_ms,0,blend_radius_m)
    |   movel([0.136190, -1.307881, -2.620358, -0.784150, 1.570796, 1.706987],accel_mss,speed_ms,0,blend_radius_m)
    |   movel([0.180166, -1.295917, -2.627508, -0.788964, 1.570796, 1.750963],accel_mss,speed_ms,0,blend_radius_m)
    |   movel([0.171306, -1.341394, -2.599322, -0.771673, 1.570796, 1.742102],accel_mss,speed_ms,0,blend_radius_m)
    |   movel([0.163298, -1.383826, -2.570469, -0.758094, 1.570796, 1.734095],accel_mss,speed_ms,0,blend_radius_m)
    |   movel([0.123568, -1.393350, -2.563640, -0.755399, 1.570796, 1.694365],accel_mss,speed_ms,0,blend_radius_m)
    |   movel([0.121109, -1.393977, -2.563186, -0.755226, 1.570796, 1.691905],accel_mss,speed_ms,0,blend_radius_m)
    |   speed_ms = 0.005
    |   movel([0.121109, -1.385358, -2.559246, -0.767785, 1.570796, 1.691905],accel_mss,speed_ms,0,blend_radius_m)
    |   speed_ms = 0.040
    |   movel([0.122958, -1.387373, -2.557801, -0.767215, 1.570796, 1.693754],accel_mss,speed_ms,0,blend_radius_m)
    |   speed_ms = 0.005
    |   movel([0.122958, -1.395977, -2.561733, -0.754679, 1.570796, 1.693754],accel_mss,speed_ms,0,blend_radius_m)
    |   speed_ms = 0.030
    |   movel([0.128656, -1.394520, -2.562792, -0.755077, 1.570796, 1.699453],accel_mss,speed_ms,0,blend_radius_m)
    |   movel([0.136033, -1.392505, -2.564251, -0.755633, 1.570796, 1.706829],accel_mss,speed_ms,0,blend_radius_m)
    |   movel([0.136283, -1.392251, -2.564435, -0.755703, 1.570796, 1.707079],accel_mss,speed_ms,0,blend_radius_m)
    |   movel([0.136095, -1.392104, -2.564541, -0.755744, 1.570796, 1.706892],accel_mss,speed_ms,0,blend_radius_m)
    |   movel([0.132890, -1.392777, -2.564055, -0.755558, 1.570796, 1.703686],accel_mss,speed_ms,0,blend_radius_m)
    |   movel([0.123079, -1.395123, -2.562354, -0.754912, 1.570796, 1.693875],accel_mss,speed_ms,0,blend_radius_m)
    |   movel([0.117381, -1.396605, -2.561276, -0.754508, 1.570796, 1.688177],accel_mss,speed_ms,0,blend_radius_m)
    |   movel([0.110029, -1.398714, -2.559736, -0.753939, 1.570796, 1.680825],accel_mss,speed_ms,0,blend_radius_m)
    |   movel([0.109786, -1.398968, -2.559550, -0.753871, 1.570796, 1.680582],accel_mss,speed_ms,0,blend_radius_m)
    |   movel([0.109978, -1.399107, -2.559448, -0.753834, 1.570796, 1.680775],accel_mss,speed_ms,0,blend_radius_m)
    |   movel([0.113172, -1.398384, -2.559977, -0.754028, 1.570796, 1.683968],accel_mss,speed_ms,0,blend_radius_m)
    |   movel([0.122958, -1.395977, -2.561733, -0.754679, 1.570796, 1.693754],accel_mss,speed_ms,0,blend_radius_m)
    |   movel([0.125412, -1.395347, -2.562191, -0.754851, 1.570796, 1.696208],accel_mss,speed_ms,0,blend_radius_m)
    |   speed_ms = 0.005
    |   movel([0.125412, -1.386738, -2.558257, -0.767394, 1.570796, 1.696208],accel_mss,speed_ms,0,blend_radius_m)
    |   speed_ms = 0.040
    |   movel([0.116105, -1.391507, -2.554820, -0.766062, 1.570796, 1.686902],accel_mss,speed_ms,0,blend_radius_m)
    |   speed_ms = 0.005
    |   movel([0.116105, -1.400081, -2.558734, -0.753574, 1.570796, 1.686902],accel_mss,speed_ms,0,blend_radius_m)
    |   speed_ms = 0.030
    |   movel([0.115433, -1.400210, -2.558640, -0.753540, 1.570796, 1.686229],accel_mss,speed_ms,0,blend_radius_m)
    |   movel([0.130214, -1.396436, -2.561399, -0.754554, 1.570796, 1.701011],accel_mss,speed_ms,0,blend_radius_m)
    |   movel([0.126246, -1.397552, -2.560585, -0.754252, 1.570796, 1.697043],accel_mss,speed_ms,0,blend_radius_m)
    |   movel([0.122632, -1.398472, -2.559913, -0.754004, 1.570796, 1.693428],accel_mss,speed_ms,0,blend_radius_m)
    |   movel([0.116105, -1.400081, -2.558734, -0.753574, 1.570796, 1.686902],accel_mss,speed_ms,0,blend_radius_m)
    |   movel([0.115433, -1.400210, -2.558640, -0.753540, 1.570796, 1.686229],accel_mss,speed_ms,0,blend_radius_m)
    |   movel([0.117195, -1.399751, -2.558976, -0.753662, 1.570796, 1.687991],accel_mss,speed_ms,0,blend_radius_m)
    |   speed_ms = 0.005
    |   movel([0.117195, -1.391174, -2.555061, -0.766154, 1.570796, 1.687991],accel_mss,speed_ms,0,blend_radius_m)
    |   speed_ms = 0.040
    |   movel([0.135389, -1.403192, -2.546259, -0.762939, 1.570796, 1.706186],accel_mss,speed_ms,0,blend_radius_m)
    |   speed_ms = 0.005
    |   movel([0.135389, -1.411681, -2.550123, -0.750585, 1.570796, 1.706186],accel_mss,speed_ms,0,blend_radius_m)
    |   speed_ms = 0.030
    |   movel([0.132351, -1.411571, -2.550206, -0.750612, 1.570796, 1.703147],accel_mss,speed_ms,0,blend_radius_m)
    |   movel([0.129158, -1.411834, -2.550008, -0.750547, 1.570796, 1.699955],accel_mss,speed_ms,0,blend_radius_m)
    |   movel([0.124985, -1.412523, -2.549490, -0.750376, 1.570796, 1.695781],accel_mss,speed_ms,0,blend_radius_m)
    |   movel([0.120763, -1.413449, -2.548793, -0.750147, 1.570796, 1.691560],accel_mss,speed_ms,0,blend_radius_m)
    |   movel([0.116520, -1.414601, -2.547924, -0.749864, 1.570796, 1.687316],accel_mss,speed_ms,0,blend_radius_m)
    |   movel([0.112269, -1.415978, -2.546882, -0.749528, 1.570796, 1.683065],accel_mss,speed_ms,0,blend_radius_m)
    |   movel([0.108963, -1.417307, -2.545875, -0.749207, 1.570796, 1.679759],accel_mss,speed_ms,0,blend_radius_m)
    |   movel([0.105717, -1.418952, -2.544624, -0.748813, 1.570796, 1.676514],accel_mss,speed_ms,0,blend_radius_m)
    |   movel([0.104975, -1.419421, -2.544266, -0.748702, 1.570796, 1.675771],accel_mss,speed_ms,0,blend_radius_m)
    |   movel([0.104579, -1.419823, -2.543960, -0.748606, 1.570796, 1.675375],accel_mss,speed_ms,0,blend_radius_m)
    |   movel([0.104380, -1.420297, -2.543598, -0.748494, 1.570796, 1.675176],accel_mss,speed_ms,0,blend_radius_m)
    |   movel([0.104317, -1.421023, -2.543043, -0.748323, 1.570796, 1.675113],accel_mss,speed_ms,0,blend_radius_m)
    |   movel([0.104506, -1.421816, -2.542436, -0.748137, 1.570796, 1.675302],accel_mss,speed_ms,0,blend_radius_m)
    |   movel([0.104722, -1.421990, -2.542302, -0.748096, 1.570796, 1.675519],accel_mss,speed_ms,0,blend_radius_m)
    |   movel([0.105057, -1.422008, -2.542289, -0.748092, 1.570796, 1.675853],accel_mss,speed_ms,0,blend_radius_m)
    |   movel([0.106352, -1.421639, -2.542572, -0.748179, 1.570796, 1.677149],accel_mss,speed_ms,0,blend_radius_m)
    |   movel([0.113761, -1.418859, -2.544695, -0.748836, 1.570796, 1.684557],accel_mss,speed_ms,0,blend_radius_m)
    |   movel([0.116206, -1.418099, -2.545273, -0.749017, 1.570796, 1.687002],accel_mss,speed_ms,0,blend_radius_m)
    |   movel([0.122098, -1.416585, -2.546423, -0.749381, 1.570796, 1.692894],accel_mss,speed_ms,0,blend_radius_m)
    |   movel([0.127857, -1.415450, -2.547282, -0.749657, 1.570796, 1.698653],accel_mss,speed_ms,0,blend_radius_m)
    |   movel([0.130091, -1.415142, -2.547515, -0.749732, 1.570796, 1.700887],accel_mss,speed_ms,0,blend_radius_m)
    |   movel([0.132283, -1.414976, -2.547641, -0.749772, 1.570796, 1.703079],accel_mss,speed_ms,0,blend_radius_m)
    |   movel([0.135410, -1.414677, -2.547866, -0.749845, 1.570796, 1.706207],accel_mss,speed_ms,0,blend_radius_m)
    |   movel([0.135692, -1.414559, -2.547956, -0.749874, 1.570796, 1.706488],accel_mss,speed_ms,0,blend_radius_m)
    |   movel([0.136035, -1.413991, -2.548384, -0.750014, 1.570796, 1.706831],accel_mss,speed_ms,0,blend_radius_m)
    |   movel([0.136292, -1.413032, -2.549107, -0.750250, 1.570796, 1.707088],accel_mss,speed_ms,0,blend_radius_m)
    |   movel([0.136326, -1.412434, -2.549557, -0.750398, 1.570796, 1.707122],accel_mss,speed_ms,0,blend_radius_m)
    |   movel([0.136203, -1.412040, -2.549853, -0.750496, 1.570796, 1.706999],accel_mss,speed_ms,0,blend_radius_m)
    |   movel([0.135900, -1.411803, -2.550031, -0.750555, 1.570796, 1.706696],accel_mss,speed_ms,0,blend_radius_m)
    |   movel([0.135389, -1.411681, -2.550123, -0.750585, 1.570796, 1.706186],accel_mss,speed_ms,0,blend_radius_m)
    |   movel([0.133194, -1.411600, -2.550184, -0.750605, 1.570796, 1.703990],accel_mss,speed_ms,0,blend_radius_m)
    |   speed_ms = 0.005
    |   movel([0.133194, -1.403110, -2.546320, -0.762960, 1.570796, 1.703990],accel_mss,speed_ms,0,blend_radius_m)
    |   speed_ms = 0.040
    |   movel([0.138194, -1.418799, -2.534513, -0.759078, 1.570796, 1.708991],accel_mss,speed_ms,0,blend_radius_m)
    |   speed_ms = 0.005
    |   movel([0.138194, -1.427173, -2.538310, -0.746905, 1.570796, 1.708991],accel_mss,speed_ms,0,blend_radius_m)
    |   speed_ms = 0.030
    |   movel([0.138358, -1.427896, -2.537751, -0.746743, 1.570796, 1.709154],accel_mss,speed_ms,0,blend_radius_m)
    |   movel([0.138370, -1.428681, -2.537141, -0.746567, 1.570796, 1.709167],accel_mss,speed_ms,0,blend_radius_m)
    |   movel([0.138233, -1.429507, -2.536500, -0.746382, 1.570796, 1.709030],accel_mss,speed_ms,0,blend_radius_m)
    |   movel([0.137950, -1.430355, -2.535840, -0.746194, 1.570796, 1.708747],accel_mss,speed_ms,0,blend_radius_m)
    |   movel([0.137520, -1.431226, -2.535161, -0.746002, 1.570796, 1.708316],accel_mss,speed_ms,0,blend_radius_m)
    |   movel([0.136968, -1.432077, -2.534496, -0.745816, 1.570796, 1.707765],accel_mss,speed_ms,0,blend_radius_m)
    |   movel([0.136306, -1.432892, -2.533858, -0.745638, 1.570796, 1.707102],accel_mss,speed_ms,0,blend_radius_m)
    |   movel([0.135547, -1.433656, -2.533260, -0.745473, 1.570796, 1.706343],accel_mss,speed_ms,0,blend_radius_m)
    |   movel([0.134679, -1.434374, -2.532697, -0.745318, 1.570796, 1.705475],accel_mss,speed_ms,0,blend_radius_m)
    |   movel([0.133750, -1.435012, -2.532196, -0.745181, 1.570796, 1.704546],accel_mss,speed_ms,0,blend_radius_m)
    |   movel([0.132774, -1.435557, -2.531768, -0.745065, 1.570796, 1.703570],accel_mss,speed_ms,0,blend_radius_m)
    |   movel([0.131774, -1.435996, -2.531421, -0.744971, 1.570796, 1.702570],accel_mss,speed_ms,0,blend_radius_m)
    |   movel([0.130764, -1.436328, -2.531160, -0.744901, 1.570796, 1.701560],accel_mss,speed_ms,0,blend_radius_m)
    |   movel([0.129766, -1.436539, -2.530994, -0.744856, 1.570796, 1.700562],accel_mss,speed_ms,0,blend_radius_m)
    |   movel([0.128797, -1.436630, -2.530922, -0.744837, 1.570796, 1.699593],accel_mss,speed_ms,0,blend_radius_m)
    |   movel([0.127878, -1.436599, -2.530947, -0.744843, 1.570796, 1.698675],accel_mss,speed_ms,0,blend_radius_m)
    |   movel([0.126988, -1.436433, -2.531078, -0.744879, 1.570796, 1.697785],accel_mss,speed_ms,0,blend_radius_m)
    |   movel([0.126197, -1.436128, -2.531318, -0.744943, 1.570796, 1.696993],accel_mss,speed_ms,0,blend_radius_m)
    |   movel([0.125516, -1.435692, -2.531661, -0.745036, 1.570796, 1.696313],accel_mss,speed_ms,0,blend_radius_m)
    |   movel([0.124968, -1.435136, -2.532098, -0.745154, 1.570796, 1.695764],accel_mss,speed_ms,0,blend_radius_m)
    |   movel([0.124576, -1.434487, -2.532608, -0.745294, 1.570796, 1.695372],accel_mss,speed_ms,0,blend_radius_m)
    |   movel([0.124345, -1.433739, -2.533195, -0.745455, 1.570796, 1.695142],accel_mss,speed_ms,0,blend_radius_m)
    |   movel([0.124284, -1.432914, -2.533842, -0.745634, 1.570796, 1.695080],accel_mss,speed_ms,0,blend_radius_m)
    |   movel([0.124391, -1.432032, -2.534532, -0.745826, 1.570796, 1.695187],accel_mss,speed_ms,0,blend_radius_m)
    |   movel([0.124667, -1.431113, -2.535249, -0.746027, 1.570796, 1.695464],accel_mss,speed_ms,0,blend_radius_m)
    |   movel([0.125101, -1.430187, -2.535971, -0.746231, 1.570796, 1.695898],accel_mss,speed_ms,0,blend_radius_m)
    |   movel([0.125686, -1.429278, -2.536678, -0.746433, 1.570796, 1.696483],accel_mss,speed_ms,0,blend_radius_m)
    |   movel([0.126405, -1.428408, -2.537353, -0.746628, 1.570796, 1.697201],accel_mss,speed_ms,0,blend_radius_m)
    |   movel([0.127256, -1.427578, -2.537997, -0.746814, 1.570796, 1.698052],accel_mss,speed_ms,0,blend_radius_m)
    |   movel([0.128199, -1.426825, -2.538580, -0.746984, 1.570796, 1.698995],accel_mss,speed_ms,0,blend_radius_m)
    |   movel([0.129210, -1.426169, -2.539087, -0.747133, 1.570796, 1.700007],accel_mss,speed_ms,0,blend_radius_m)
    |   movel([0.130268, -1.425626, -2.539506, -0.747257, 1.570796, 1.701064],accel_mss,speed_ms,0,blend_radius_m)
    |   movel([0.131525, -1.425159, -2.539866, -0.747363, 1.570796, 1.702321],accel_mss,speed_ms,0,blend_radius_m)
    |   movel([0.132767, -1.424897, -2.540069, -0.747424, 1.570796, 1.703563],accel_mss,speed_ms,0,blend_radius_m)
    |   movel([0.134027, -1.424827, -2.540123, -0.747440, 1.570796, 1.704823],accel_mss,speed_ms,0,blend_radius_m)
    |   movel([0.135198, -1.424949, -2.540028, -0.747412, 1.570796, 1.705994],accel_mss,speed_ms,0,blend_radius_m)
    |   movel([0.136238, -1.425259, -2.539790, -0.747341, 1.570796, 1.707034],accel_mss,speed_ms,0,blend_radius_m)
    |   movel([0.137130, -1.425751, -2.539409, -0.747228, 1.570796, 1.707926],accel_mss,speed_ms,0,blend_radius_m)
    |   movel([0.137776, -1.426377, -2.538926, -0.747086, 1.570796, 1.708572],accel_mss,speed_ms,0,blend_radius_m)
    |   movel([0.138194, -1.427173, -2.538310, -0.746905, 1.570796, 1.708991],accel_mss,speed_ms,0,blend_radius_m)
    |   movel([0.138358, -1.427896, -2.537751, -0.746743, 1.570796, 1.709154],accel_mss,speed_ms,0,blend_radius_m)
    |   movel([0.138370, -1.428681, -2.537141, -0.746567, 1.570796, 1.709167],accel_mss,speed_ms,0,blend_radius_m)
    |   movel([0.138305, -1.429072, -2.536838, -0.746479, 1.570796, 1.709102],accel_mss,speed_ms,0,blend_radius_m)
    |   speed_ms = 0.005
    |   movel([0.138305, -1.420712, -2.533048, -0.758629, 1.570796, 1.709102],accel_mss,speed_ms,0,blend_radius_m)
    |   speed_ms = 0.040
    |   movel([0.134556, -1.420607, -2.533129, -0.758654, 1.570796, 1.705352],accel_mss,speed_ms,0,blend_radius_m)
    |   speed_ms = 0.005
    |   movel([0.134556, -1.428968, -2.536919, -0.746503, 1.570796, 1.705352],accel_mss,speed_ms,0,blend_radius_m)
    |   speed_ms = 0.030
    |   movel([0.133917, -1.428271, -2.537460, -0.746658, 1.570796, 1.704714],accel_mss,speed_ms,0,blend_radius_m)
    |   movel([0.133441, -1.427977, -2.537688, -0.746724, 1.570796, 1.704237],accel_mss,speed_ms,0,blend_radius_m)
    |   movel([0.132234, -1.427638, -2.537950, -0.746801, 1.570796, 1.703030],accel_mss,speed_ms,0,blend_radius_m)
    |   movel([0.131729, -1.427666, -2.537929, -0.746794, 1.570796, 1.702526],accel_mss,speed_ms,0,blend_radius_m)
    |   movel([0.131197, -1.427878, -2.537765, -0.746747, 1.570796, 1.701993],accel_mss,speed_ms,0,blend_radius_m)
    |   movel([0.130376, -1.428385, -2.537371, -0.746633, 1.570796, 1.701173],accel_mss,speed_ms,0,blend_radius_m)
    |   movel([0.129437, -1.429129, -2.536794, -0.746467, 1.570796, 1.700234],accel_mss,speed_ms,0,blend_radius_m)
    |   movel([0.128656, -1.429994, -2.536121, -0.746274, 1.570796, 1.699452],accel_mss,speed_ms,0,blend_radius_m)
    |   movel([0.128121, -1.430888, -2.535424, -0.746077, 1.570796, 1.698917],accel_mss,speed_ms,0,blend_radius_m)
    |   movel([0.127854, -1.431785, -2.534724, -0.745880, 1.570796, 1.698650],accel_mss,speed_ms,0,blend_radius_m)
    |   movel([0.127885, -1.432564, -2.534115, -0.745709, 1.570796, 1.698681],accel_mss,speed_ms,0,blend_radius_m)
    |   movel([0.128207, -1.433198, -2.533619, -0.745572, 1.570796, 1.699003],accel_mss,speed_ms,0,blend_radius_m)
    |   movel([0.128793, -1.433633, -2.533279, -0.745478, 1.570796, 1.699589],accel_mss,speed_ms,0,blend_radius_m)
    |   movel([0.129581, -1.433830, -2.533124, -0.745435, 1.570796, 1.700377],accel_mss,speed_ms,0,blend_radius_m)
    |   movel([0.130539, -1.433772, -2.533170, -0.745448, 1.570796, 1.701335],accel_mss,speed_ms,0,blend_radius_m)
    |   movel([0.131550, -1.433464, -2.533411, -0.745514, 1.570796, 1.702346],accel_mss,speed_ms,0,blend_radius_m)
    |   movel([0.132541, -1.432926, -2.533832, -0.745631, 1.570796, 1.703337],accel_mss,speed_ms,0,blend_radius_m)
    |   movel([0.133429, -1.432211, -2.534392, -0.745787, 1.570796, 1.704225],accel_mss,speed_ms,0,blend_radius_m)
    |   movel([0.134112, -1.431393, -2.535031, -0.745966, 1.570796, 1.704908],accel_mss,speed_ms,0,blend_radius_m)
    |   movel([0.134561, -1.430517, -2.535713, -0.746158, 1.570796, 1.705357],accel_mss,speed_ms,0,blend_radius_m)
    |   movel([0.134713, -1.429691, -2.536357, -0.746341, 1.570796, 1.705509],accel_mss,speed_ms,0,blend_radius_m)
    |   movel([0.134556, -1.428968, -2.536919, -0.746503, 1.570796, 1.705352],accel_mss,speed_ms,0,blend_radius_m)
    |   movel([0.133917, -1.428271, -2.537460, -0.746658, 1.570796, 1.704714],accel_mss,speed_ms,0,blend_radius_m)
    |   movel([0.133441, -1.427977, -2.537688, -0.746724, 1.570796, 1.704237],accel_mss,speed_ms,0,blend_radius_m)
    |   movel([0.133153, -1.427897, -2.537750, -0.746742, 1.570796, 1.703949],accel_mss,speed_ms,0,blend_radius_m)
    |   speed_ms = 0.005
    |   movel([0.133153, -1.419528, -2.533955, -0.758906, 1.570796, 1.703949],accel_mss,speed_ms,0,blend_radius_m)
    |   speed_ms = 0.040
    |   movel([0.135995, -1.422829, -2.531421, -0.758139, 1.570796, 1.706791],accel_mss,speed_ms,0,blend_radius_m)
    |   speed_ms = 0.005
    |   movel([0.135995, -1.431173, -2.535202, -0.746014, 1.570796, 1.706791],accel_mss,speed_ms,0,blend_radius_m)
    |   speed_ms = 0.030
    |   movel([0.134998, -1.432565, -2.534115, -0.745709, 1.570796, 1.705795],accel_mss,speed_ms,0,blend_radius_m)
    |   movel([0.134437, -1.433135, -2.533669, -0.745586, 1.570796, 1.705233],accel_mss,speed_ms,0,blend_radius_m)
    |   movel([0.133806, -1.433638, -2.533275, -0.745477, 1.570796, 1.704602],accel_mss,speed_ms,0,blend_radius_m)
    |   movel([0.133094, -1.434081, -2.532927, -0.745381, 1.570796, 1.703890],accel_mss,speed_ms,0,blend_radius_m)
    |   movel([0.132350, -1.434430, -2.532653, -0.745306, 1.570796, 1.703146],accel_mss,speed_ms,0,blend_radius_m)
    |   movel([0.130573, -1.434990, -2.532213, -0.745186, 1.570796, 1.701369],accel_mss,speed_ms,0,blend_radius_m)
    |   movel([0.129278, -1.435172, -2.532070, -0.745147, 1.570796, 1.700074],accel_mss,speed_ms,0,blend_radius_m)
    |   movel([0.128073, -1.435109, -2.532120, -0.745160, 1.570796, 1.698870],accel_mss,speed_ms,0,blend_radius_m)
    |   movel([0.127106, -1.434798, -2.532364, -0.745227, 1.570796, 1.697902],accel_mss,speed_ms,0,blend_radius_m)
    |   movel([0.126370, -1.434228, -2.532812, -0.745349, 1.570796, 1.697166],accel_mss,speed_ms,0,blend_radius_m)
    |   movel([0.125934, -1.433457, -2.533416, -0.745516, 1.570796, 1.696730],accel_mss,speed_ms,0,blend_radius_m)
    |   movel([0.125816, -1.432515, -2.534154, -0.745720, 1.570796, 1.696612],accel_mss,speed_ms,0,blend_radius_m)
    |   movel([0.126013, -1.431433, -2.534999, -0.745957, 1.570796, 1.696809],accel_mss,speed_ms,0,blend_radius_m)
    |   movel([0.126501, -1.430319, -2.535868, -0.746202, 1.570796, 1.697298],accel_mss,speed_ms,0,blend_radius_m)
    |   movel([0.126929, -1.429665, -2.536377, -0.746347, 1.570796, 1.697725],accel_mss,speed_ms,0,blend_radius_m)
    |   movel([0.127449, -1.429040, -2.536862, -0.746486, 1.570796, 1.698245],accel_mss,speed_ms,0,blend_radius_m)
    |   movel([0.128048, -1.428461, -2.537312, -0.746616, 1.570796, 1.698845],accel_mss,speed_ms,0,blend_radius_m)
    |   movel([0.128715, -1.427941, -2.537715, -0.746732, 1.570796, 1.699511],accel_mss,speed_ms,0,blend_radius_m)
    |   movel([0.130262, -1.427050, -2.538405, -0.746933, 1.570796, 1.701059],accel_mss,speed_ms,0,blend_radius_m)
    |   movel([0.131068, -1.426723, -2.538659, -0.747007, 1.570796, 1.701864],accel_mss,speed_ms,0,blend_radius_m)
    |   movel([0.132662, -1.426332, -2.538961, -0.747096, 1.570796, 1.703458],accel_mss,speed_ms,0,blend_radius_m)
    |   movel([0.133426, -1.426276, -2.539004, -0.747109, 1.570796, 1.704223],accel_mss,speed_ms,0,blend_radius_m)
    |   movel([0.134822, -1.426449, -2.538871, -0.747069, 1.570796, 1.705618],accel_mss,speed_ms,0,blend_radius_m)
    |   movel([0.135381, -1.426668, -2.538701, -0.747020, 1.570796, 1.706178],accel_mss,speed_ms,0,blend_radius_m)
    |   movel([0.135852, -1.426987, -2.538455, -0.746948, 1.570796, 1.706648],accel_mss,speed_ms,0,blend_radius_m)
    |   movel([0.136224, -1.427393, -2.538140, -0.746856, 1.570796, 1.707020],accel_mss,speed_ms,0,blend_radius_m)
    |   movel([0.136811, -1.428844, -2.537015, -0.746530, 1.570796, 1.707608],accel_mss,speed_ms,0,blend_radius_m)
    |   movel([0.136842, -1.429394, -2.536587, -0.746407, 1.570796, 1.707638],accel_mss,speed_ms,0,blend_radius_m)
    |   movel([0.136640, -1.429996, -2.536119, -0.746274, 1.570796, 1.707437],accel_mss,speed_ms,0,blend_radius_m)
    |   movel([0.135995, -1.431173, -2.535202, -0.746014, 1.570796, 1.706791],accel_mss,speed_ms,0,blend_radius_m)
    |   movel([0.134998, -1.432565, -2.534115, -0.745709, 1.570796, 1.705795],accel_mss,speed_ms,0,blend_radius_m)
    |   movel([0.134437, -1.433135, -2.533669, -0.745586, 1.570796, 1.705233],accel_mss,speed_ms,0,blend_radius_m)
    |   speed_ms = 0.005
    |   movel([0.134437, -1.424805, -2.529896, -0.757687, 1.570796, 1.705233],accel_mss,speed_ms,0,blend_radius_m)
    |   speed_ms = 0.040
    |   movel([0.151093, -1.420110, -2.533510, -0.758770, 1.570796, 1.721889],accel_mss,speed_ms,0,blend_radius_m)
    |   speed_ms = 0.005
    |   movel([0.151093, -1.428474, -2.537302, -0.746613, 1.570796, 1.721889],accel_mss,speed_ms,0,blend_radius_m)
    |   speed_ms = 0.030
    |   movel([0.152972, -1.428072, -2.537614, -0.746703, 1.570796, 1.723768],accel_mss,speed_ms,0,blend_radius_m)
    |   movel([0.154140, -1.421471, -2.542700, -0.748218, 1.570796, 1.724936],accel_mss,speed_ms,0,blend_radius_m)
    |   movel([0.155326, -1.414805, -2.547770, -0.749814, 1.570796, 1.726122],accel_mss,speed_ms,0,blend_radius_m)
